LIN {X 0,Y 736.002,Z 322.542,A -85,B 0,C 180,E1 27536.573,E2 27536.573} C_VEL
LIN {X 0,Y 736.007,Z 322.537,A -85,B 0,C 180,E1 27534.23,E2 27534.23} C_VEL
LIN {X 0,Y 736.096,Z 322.542,A -85,B 0,C 180,E1 27531.444,E2 27531.444} C_VEL
LIN {X 0,Y 736.087,Z 322.537,A -85,B 0,C 180,E1 27529.14,E2 27529.14} C_VEL
LIN {X 0,Y 735.045,Z 322.662,A -85,B 0,C 180,E1 27528.541,E2 27528.541} C_VEL
LIN {X 0,Y 728.618,Z 323.468,A -85,B 0,C 180,E1 27526.861,E2 27526.861} C_VEL
LIN {X 0,Y 728.077,Z 323.53,A -85,B 0,C 180,E1 27526.425,E2 27526.425} C_VEL
LIN {X 0,Y 728.078,Z 323.523,A -85,B 0,C 180,E1 27524.01,E2 27524.01} C_VEL
LIN {X 0,Y 728.156,Z 323.53,A -85,B 0,C 180,E1 27521.257,E2 27521.257} C_VEL
LIN {X 0,Y 728.092,Z 323.528,A -85,B 0,C 180,E1 27518.389,E2 27518.389} C_VEL
LIN {X 0,Y 728.082,Z 323.529,A -85,B 0,C 180,E1 27515.928,E2 27515.928} C_VEL
LIN {X 0,Y 728.15,Z 323.533,A -85,B 0,C 180,E1 27513.196,E2 27513.196} C_VEL
LIN {X 0,Y 728.1,Z 323.527,A -85,B 0,C 180,E1 27510.215,E2 27510.215} C_VEL
LIN {X 0,Y 728.091,Z 323.531,A -85,B 0,C 180,E1 27507.709,E2 27507.709} C_VEL
LIN {X 0,Y 728.156,Z 323.534,A -85,B 0,C 180,E1 27504.925,E2 27504.925} C_VEL
LIN {X 0,Y 728.109,Z 323.531,A -85,B 0,C 180,E1 27502.021,E2 27502.021} C_VEL
LIN {X 0,Y 728.178,Z 323.766,A -85,B 0,C 180,E1 27500.292,E2 27500.292} C_VEL
LIN {X 0,Y 729.309,Z 326.852,A -85,B 0,C 180,E1 27499.984,E2 27499.984} C_VEL
LIN {X 0,Y 733.452,Z 336.015,A -85,B 0,C 180,E1 27499.025,E2 27499.025} C_VEL
LIN {X 0,Y 733.504,Z 341.36,A -85,B 0,C 180,E1 27498.676,E2 27498.676} C_VEL
LIN {X 0,Y 735.856,Z 350.593,A -85,B 0,C 180,E1 27498.388,E2 27498.388} C_VEL
LIN {X 0,Y 734.928,Z 566.12,A -85,B 0,C 180,E1 27495.714,E2 27495.714} C_VEL
LIN {X 0,Y 734.028,Z 793.03,A -85,B 0,C 180,E1 27492.997,E2 27492.997} C_VEL
LIN {X 0,Y 733.826,Z 825.795,A -85,B 0,C 180,E1 27492.567,E2 27492.567} C_VEL
LIN {X 0,Y 733.495,Z 853.318,A -85,B 0,C 180,E1 27492.041,E2 27492.041} C_VEL
LIN {X 0,Y 733.131,Z 879.099,A -85,B 0,C 180,E1 27491.393,E2 27491.393} C_VEL
LIN {X 0,Y 732.64,Z 907.823,A -85,B 0,C 180,E1 27490.487,E2 27490.487} C_VEL
LIN {X 0,Y 732.19,Z 930.681,A -85,B 0,C 180,E1 27489.622,E2 27489.622} C_VEL
LIN {X 0,Y 731.795,Z 951.079,A -85,B 0,C 180,E1 27488.739,E2 27488.739} C_VEL
LIN {X 0,Y 731.381,Z 971.985,A -85,B 0,C 180,E1 27487.718,E2 27487.718} C_VEL
LIN {X 0,Y 730.845,Z 997.329,A -85,B 0,C 180,E1 27486.309,E2 27486.309} C_VEL
LIN {X 0,Y 730.379,Z 1017.32,A -85,B 0,C 180,E1 27485.048,E2 27485.048} C_VEL
LIN {X 0,Y 730.011,Z 1035.431,A -85,B 0,C 180,E1 27483.785,E2 27483.785} C_VEL
LIN {X 0,Y 729.644,Z 1055.852,A -85,B 0,C 180,E1 27482.213,E2 27482.213} C_VEL
LIN {X 0,Y 729.213,Z 1074.861,A -85,B 0,C 180,E1 27480.558,E2 27480.558} C_VEL
LIN {X 0,Y 728.957,Z 1090.57,A -85,B 0,C 180,E1 27479.049,E2 27479.049} C_VEL
LIN {X 0,Y 728.689,Z 1108.03,A -85,B 0,C 180,E1 27477.189,E2 27477.189} C_VEL
LIN {X 0,Y 728.436,Z 1123.152,A -85,B 0,C 180,E1 27475.357,E2 27475.357} C_VEL
LIN {X 0,Y 728.291,Z 1134.68,A -85,B 0,C 180,E1 27473.805,E2 27473.805} C_VEL
LIN {X 0,Y 728.159,Z 1145.498,A -85,B 0,C 180,E1 27472.186,E2 27472.186} C_VEL
LIN {X 0,Y 728.088,Z 1156.487,A -85,B 0,C 180,E1 27470.331,E2 27470.331} C_VEL
LIN {X 0,Y 727.975,Z 1167.358,A -85,B 0,C 180,E1 27468.166,E2 27468.166} C_VEL
LIN {X 0,Y 727.957,Z 1175.727,A -85,B 0,C 180,E1 27466.19,E2 27466.19} C_VEL
LIN {X 0,Y 727.928,Z 1182.921,A -85,B 0,C 180,E1 27464.071,E2 27464.071} C_VEL
LIN {X 0,Y 727.913,Z 1188.371,A -85,B 0,C 180,E1 27461.971,E2 27461.971} C_VEL
LIN {X 0,Y 727.907,Z 1192.173,A -85,B 0,C 180,E1 27459.887,E2 27459.887} C_VEL
LIN {X 0,Y 727.904,Z 1194.402,A -85,B 0,C 180,E1 27457.736,E2 27457.736} C_VEL
LIN {X 0,Y 727.892,Z 1194.882,A -85,B 0,C 180,E1 27455.518,E2 27455.518} C_VEL
LIN {X 0,Y 727.906,Z 1193.93,A -85,B 0,C 180,E1 27453.544,E2 27453.544} C_VEL
LIN {X 0,Y 727.907,Z 1191.228,A -85,B 0,C 180,E1 27451.416,E2 27451.416} C_VEL
LIN {X 0,Y 727.917,Z 1187.057,A -85,B 0,C 180,E1 27449.37,E2 27449.37} C_VEL
LIN {X 0,Y 727.937,Z 1181.082,A -85,B 0,C 180,E1 27447.244,E2 27447.244} C_VEL
LIN {X 0,Y 727.952,Z 1173.342,A -85,B 0,C 180,E1 27445.114,E2 27445.114} C_VEL
LIN {X 0,Y 728.022,Z 1163.33,A -85,B 0,C 180,E1 27442.899,E2 27442.899} C_VEL
LIN {X 0,Y 728.076,Z 1154.04,A -85,B 0,C 180,E1 27441.152,E2 27441.152} C_VEL
LIN {X 0,Y 728.191,Z 1144.427,A -85,B 0,C 180,E1 27439.557,E2 27439.557} C_VEL
LIN {X 0,Y 728.307,Z 1133.054,A -85,B 0,C 180,E1 27437.874,E2 27437.874} C_VEL
LIN {X 0,Y 728.521,Z 1117.682,A -85,B 0,C 180,E1 27435.859,E2 27435.859} C_VEL
LIN {X 0,Y 728.753,Z 1102.122,A -85,B 0,C 180,E1 27434.073,E2 27434.073} C_VEL
LIN {X 0,Y 728.985,Z 1087.151,A -85,B 0,C 180,E1 27432.519,E2 27432.519} C_VEL
LIN {X 0,Y 729.387,Z 1068.169,A -85,B 0,C 180,E1 27430.745,E2 27430.745} C_VEL
LIN {X 0,Y 729.694,Z 1049.723,A -85,B 0,C 180,E1 27429.212,E2 27429.212} C_VEL
LIN {X 0,Y 730.068,Z 1032.568,A -85,B 0,C 180,E1 27427.917,E2 27427.917} C_VEL
LIN {X 0,Y 730.59,Z 1011.035,A -85,B 0,C 180,E1 27426.445,E2 27426.445} C_VEL
LIN {X 0,Y 731.026,Z 987.732,A -85,B 0,C 180,E1 27425.046,E2 27425.046} C_VEL
LIN {X 0,Y 731.424,Z 968.525,A -85,B 0,C 180,E1 27424.015,E2 27424.015} C_VEL
LIN {X 0,Y 731.828,Z 948.858,A -85,B 0,C 180,E1 27423.069,E2 27423.069} C_VEL
LIN {X 0,Y 732.349,Z 925.446,A -85,B 0,C 180,E1 27422.076,E2 27422.076} C_VEL
LIN {X 0,Y 732.817,Z 899.396,A -85,B 0,C 180,E1 27421.14,E2 27421.14} C_VEL
LIN {X 0,Y 733.19,Z 875.306,A -85,B 0,C 180,E1 27420.412,E2 27420.412} C_VEL
LIN {X 0,Y 733.552,Z 848.854,A -85,B 0,C 180,E1 27419.773,E2 27419.773} C_VEL
LIN {X 0,Y 733.842,Z 821.735,A -85,B 0,C 180,E1 27419.281,E2 27419.281} C_VEL
LIN {X 0,Y 734.101,Z 774.815,A -85,B 0,C 180,E1 27418.699,E2 27418.699} C_VEL
LIN {X 0,Y 734.997,Z 548.599,A -85,B 0,C 180,E1 27415.982,E2 27415.982} C_VEL
LIN {X 0,Y 735.843,Z 349.755,A -85,B 0,C 180,E1 27413.511,E2 27413.511} C_VEL
LIN {X 0,Y 733.426,Z 340.384,A -85,B 0,C 180,E1 27413.189,E2 27413.189} C_VEL
LIN {X 0,Y 733.459,Z 336.113,A -85,B 0,C 180,E1 27412.893,E2 27412.893} C_VEL
LIN {X 0,Y 729.199,Z 326.593,A -85,B 0,C 180,E1 27411.9,E2 27411.9} C_VEL
LIN {X 0,Y 728.144,Z 323.532,A -85,B 0,C 180,E1 27411.584,E2 27411.584} C_VEL
LIN {X 0,Y 728.135,Z 323.53,A -85,B 0,C 180,E1 27408.691,E2 27408.691} C_VEL
LIN {X 0,Y 728.16,Z 323.524,A -85,B 0,C 180,E1 27405.768,E2 27405.768} C_VEL
LIN {X 0,Y 728.142,Z 323.533,A -85,B 0,C 180,E1 27402.716,E2 27402.716} C_VEL
LIN {X 0,Y 728.143,Z 323.524,A -85,B 0,C 180,E1 27399.786,E2 27399.786} C_VEL
LIN {X 0,Y 728.147,Z 323.533,A -85,B 0,C 180,E1 27396.68,E2 27396.68} C_VEL
LIN {X 0,Y 728.122,Z 323.525,A -85,B 0,C 180,E1 27393.819,E2 27393.819} C_VEL
LIN {X 0,Y 728.156,Z 323.531,A -85,B 0,C 180,E1 27390.882,E2 27390.882} C_VEL
LIN {X 0,Y 728.109,Z 323.526,A -85,B 0,C 180,E1 27388.101,E2 27388.101} C_VEL
LIN {X 0,Y 728.139,Z 323.518,A -85,B 0,C 180,E1 27385.369,E2 27385.369} C_VEL
LIN {X 0,Y 728.122,Z 323.528,A -85,B 0,C 180,E1 27382.273,E2 27382.273} C_VEL
LIN {X 0,Y 728.103,Z 323.52,A -85,B 0,C 180,E1 27379.578,E2 27379.578} C_VEL
LIN {X 0,Y 728.159,Z 323.529,A -85,B 0,C 180,E1 27376.678,E2 27376.678} C_VEL
LIN {X 0,Y 728.096,Z 323.52,A -85,B 0,C 180,E1 27373.854,E2 27373.854} C_VEL
LIN {X 0,Y 728.105,Z 323.526,A -85,B 0,C 180,E1 27371.245,E2 27371.245} C_VEL
LIN {X 0,Y 728.138,Z 323.533,A -85,B 0,C 180,E1 27368.211,E2 27368.211} C_VEL
LIN {X 0,Y 728.082,Z 323.528,A -85,B 0,C 180,E1 27365.517,E2 27365.517} C_VEL
LIN {X 0,Y 728.103,Z 323.528,A -85,B 0,C 180,E1 27362.991,E2 27362.991} C_VEL
LIN {X 0,Y 728.113,Z 323.533,A -85,B 0,C 180,E1 27359.921,E2 27359.921} C_VEL
LIN {X 0,Y 728.074,Z 323.531,A -85,B 0,C 180,E1 27357.402,E2 27357.402} C_VEL
LIN {X 0,Y 728.08,Z 323.529,A -85,B 0,C 180,E1 27354.958,E2 27354.958} C_VEL
LIN {X 0,Y 728.149,Z 323.531,A -85,B 0,C 180,E1 27352.028,E2 27352.028} C_VEL
LIN {X 0,Y 728.068,Z 323.532,A -85,B 0,C 180,E1 27349.315,E2 27349.315} C_VEL
LIN {X 0,Y 728.06,Z 323.525,A -85,B 0,C 180,E1 27346.983,E2 27346.983} C_VEL
LIN {X 0,Y 728.083,Z 323.529,A -85,B 0,C 180,E1 27344.548,E2 27344.548} C_VEL
LIN {X 0,Y 728.077,Z 323.527,A -85,B 0,C 180,E1 27341.421,E2 27341.421} C_VEL
LIN {X 0,Y 728.05,Z 323.531,A -85,B 0,C 180,E1 27338.995,E2 27338.995} C_VEL
LIN {X 0,Y 728.048,Z 323.534,A -85,B 0,C 180,E1 27336.749,E2 27336.749} C_VEL
LIN {X 0,Y 728.078,Z 323.524,A -85,B 0,C 180,E1 27334.276,E2 27334.276} C_VEL
LIN {X 0,Y 728.074,Z 323.533,A -85,B 0,C 180,E1 27331.181,E2 27331.181} C_VEL
LIN {X 0,Y 728.057,Z 323.531,A -85,B 0,C 180,E1 27328.818,E2 27328.818} C_VEL
LIN {X 0,Y 728.061,Z 323.534,A -85,B 0,C 180,E1 27326.472,E2 27326.472} C_VEL
LIN {X 0,Y 728.129,Z 323.535,A -85,B 0,C 180,E1 27323.808,E2 27323.808} C_VEL
LIN {X 0,Y 728.083,Z 323.535,A -85,B 0,C 180,E1 27320.888,E2 27320.888} C_VEL
LIN {X 0,Y 728.069,Z 323.533,A -85,B 0,C 180,E1 27318.446,E2 27318.446} C_VEL
LIN {X 0,Y 728.093,Z 323.537,A -85,B 0,C 180,E1 27315.981,E2 27315.981} C_VEL
LIN {X 0,Y 728.144,Z 323.69,A -85,B 0,C 180,E1 27315.022,E2 27315.022} C_VEL
LIN {X 0,Y 729.555,Z 327.257,A -85,B 0,C 180,E1 27314.658,E2 27314.658} C_VEL
LIN {X 0,Y 733.674,Z 336.351,A -85,B 0,C 180,E1 27313.706,E2 27313.706} C_VEL
LIN {X 0,Y 733.608,Z 351.232,A -85,B 0,C 180,E1 27312.715,E2 27312.715} C_VEL
LIN {X 0,Y 735.832,Z 360.077,A -85,B 0,C 180,E1 27312.441,E2 27312.441} C_VEL
LIN {X 0,Y 734.945,Z 570.243,A -85,B 0,C 180,E1 27309.832,E2 27309.832} C_VEL
LIN {X 0,Y 734.062,Z 795.119,A -85,B 0,C 180,E1 27307.135,E2 27307.135} C_VEL
LIN {X 0,Y 733.838,Z 833.798,A -85,B 0,C 180,E1 27306.643,E2 27306.643} C_VEL
LIN {X 0,Y 733.521,Z 860.678,A -85,B 0,C 180,E1 27306.143,E2 27306.143} C_VEL
LIN {X 0,Y 733.18,Z 886.466,A -85,B 0,C 180,E1 27305.512,E2 27305.512} C_VEL
LIN {X 0,Y 732.754,Z 914.371,A -85,B 0,C 180,E1 27304.654,E2 27304.654} C_VEL
LIN {X 0,Y 732.218,Z 939.469,A -85,B 0,C 180,E1 27303.717,E2 27303.717} C_VEL
LIN {X 0,Y 731.801,Z 960.579,A -85,B 0,C 180,E1 27302.808,E2 27302.808} C_VEL
LIN {X 0,Y 731.386,Z 982.079,A -85,B 0,C 180,E1 27301.758,E2 27301.758} C_VEL
LIN {X 0,Y 730.853,Z 1007.148,A -85,B 0,C 180,E1 27300.366,E2 27300.366} C_VEL
LIN {X 0,Y 730.377,Z 1027.561,A -85,B 0,C 180,E1 27299.078,E2 27299.078} C_VEL
LIN {X 0,Y 729.986,Z 1046.46,A -85,B 0,C 180,E1 27297.756,E2 27297.756} C_VEL
LIN {X 0,Y 729.574,Z 1068.227,A -85,B 0,C 180,E1 27296.056,E2 27296.056} C_VEL
LIN {X 0,Y 729.193,Z 1085.444,A -85,B 0,C 180,E1 27294.55,E2 27294.55} C_VEL
LIN {X 0,Y 728.946,Z 1101.387,A -85,B 0,C 180,E1 27293.012,E2 27293.012} C_VEL
LIN {X 0,Y 728.632,Z 1120.118,A -85,B 0,C 180,E1 27290.988,E2 27290.988} C_VEL
LIN {X 0,Y 728.422,Z 1133.8,A -85,B 0,C 180,E1 27289.318,E2 27289.318} C_VEL
LIN {X 0,Y 728.291,Z 1145.415,A -85,B 0,C 180,E1 27287.746,E2 27287.746} C_VEL
LIN {X 0,Y 728.151,Z 1156.938,A -85,B 0,C 180,E1 27286.005,E2 27286.005} C_VEL
LIN {X 0,Y 728.048,Z 1169.419,A -85,B 0,C 180,E1 27283.826,E2 27283.826} C_VEL
LIN {X 0,Y 727.974,Z 1178.071,A -85,B 0,C 180,E1 27282.051,E2 27282.051} C_VEL
LIN {X 0,Y 727.953,Z 1185.836,A -85,B 0,C 180,E1 27280.206,E2 27280.206} C_VEL
LIN {X 0,Y 727.927,Z 1193.11,A -85,B 0,C 180,E1 27278.054,E2 27278.054} C_VEL
LIN {X 0,Y 727.914,Z 1198.421,A -85,B 0,C 180,E1 27275.993,E2 27275.993} C_VEL
LIN {X 0,Y 727.907,Z 1202.277,A -85,B 0,C 180,E1 27273.86,E2 27273.86} C_VEL
LIN {X 0,Y 727.908,Z 1204.493,A -85,B 0,C 180,E1 27271.653,E2 27271.653} C_VEL
LIN {X 0,Y 727.89,Z 1204.872,A -85,B 0,C 180,E1 27269.528,E2 27269.528} C_VEL
LIN {X 0,Y 727.906,Z 1203.905,A -85,B 0,C 180,E1 27267.56,E2 27267.56} C_VEL
LIN {X 0,Y 727.907,Z 1201.179,A -85,B 0,C 180,E1 27265.431,E2 27265.431} C_VEL
LIN {X 0,Y 727.916,Z 1196.957,A -85,B 0,C 180,E1 27263.375,E2 27263.375} C_VEL
LIN {X 0,Y 727.936,Z 1191.149,A -85,B 0,C 180,E1 27261.31,E2 27261.31} C_VEL
LIN {X 0,Y 727.945,Z 1183.639,A -85,B 0,C 180,E1 27259.234,E2 27259.234} C_VEL
LIN {X 0,Y 728.028,Z 1173.527,A -85,B 0,C 180,E1 27256.983,E2 27256.983} C_VEL
LIN {X 0,Y 728.084,Z 1164.528,A -85,B 0,C 180,E1 27255.282,E2 27255.282} C_VEL
LIN {X 0,Y 728.169,Z 1154.742,A -85,B 0,C 180,E1 27253.651,E2 27253.651} C_VEL
LIN {X 0,Y 728.298,Z 1144.115,A -85,B 0,C 180,E1 27252.07,E2 27252.07} C_VEL
LIN {X 0,Y 728.489,Z 1130.976,A -85,B 0,C 180,E1 27250.318,E2 27250.318} C_VEL
LIN {X 0,Y 728.741,Z 1113.473,A -85,B 0,C 180,E1 27248.264,E2 27248.264} C_VEL
LIN {X 0,Y 728.956,Z 1098.833,A -85,B 0,C 180,E1 27246.732,E2 27246.732} C_VEL
LIN {X 0,Y 729.278,Z 1082.528,A -85,B 0,C 180,E1 27245.183,E2 27245.183} C_VEL
LIN {X 0,Y 729.687,Z 1061.272,A -85,B 0,C 180,E1 27243.38,E2 27243.38} C_VEL
LIN {X 0,Y 730.037,Z 1043.447,A -85,B 0,C 180,E1 27242.025,E2 27242.025} C_VEL
LIN {X 0,Y 730.495,Z 1023.595,A -85,B 0,C 180,E1 27240.659,E2 27240.659} C_VEL
LIN {X 0,Y 731.011,Z 999.737,A -85,B 0,C 180,E1 27239.204,E2 27239.204} C_VEL
LIN {X 0,Y 731.426,Z 978.531,A -85,B 0,C 180,E1 27238.06,E2 27238.06} C_VEL
LIN {X 0,Y 731.863,Z 957.714,A -85,B 0,C 180,E1 27237.061,E2 27237.061} C_VEL
LIN {X 0,Y 732.437,Z 932.727,A -85,B 0,C 180,E1 27236.012,E2 27236.012} C_VEL
LIN {X 0,Y 732.844,Z 907.023,A -85,B 0,C 180,E1 27235.109,E2 27235.109} C_VEL
LIN {X 0,Y 733.217,Z 883.762,A -85,B 0,C 180,E1 27234.416,E2 27234.416} C_VEL
LIN {X 0,Y 733.575,Z 857.292,A -85,B 0,C 180,E1 27233.785,E2 27233.785} C_VEL
LIN {X 0,Y 733.854,Z 830.083,A -85,B 0,C 180,E1 27233.3,E2 27233.3} C_VEL
LIN {X 0,Y 734.247,Z 744.981,A -85,B 0,C 180,E1 27232.271,E2 27232.271} C_VEL
LIN {X 0,Y 735.141,Z 523.003,A -85,B 0,C 180,E1 27229.59,E2 27229.59} C_VEL
LIN {X 0,Y 735.76,Z 359.115,A -85,B 0,C 180,E1 27227.541,E2 27227.541} C_VEL
LIN {X 0,Y 733.481,Z 350.368,A -85,B 0,C 180,E1 27227.245,E2 27227.245} C_VEL
LIN {X 0,Y 733.541,Z 335.961,A -85,B 0,C 180,E1 27226.257,E2 27226.257} C_VEL
LIN {X 0,Y 728.192,Z 324.004,A -85,B 0,C 180,E1 27225.004,E2 27225.004} C_VEL
LIN {X 0,Y 728.129,Z 323.534,A -85,B 0,C 180,E1 27224.943,E2 27224.943} C_VEL
LIN {X 0,Y 728.093,Z 323.536,A -85,B 0,C 180,E1 27221.975,E2 27221.975} C_VEL
LIN {X 0,Y 728.069,Z 323.534,A -85,B 0,C 180,E1 27219.484,E2 27219.484} C_VEL
LIN {X 0,Y 728.082,Z 323.532,A -85,B 0,C 180,E1 27217.072,E2 27217.072} C_VEL
LIN {X 0,Y 728.128,Z 323.533,A -85,B 0,C 180,E1 27214.102,E2 27214.102} C_VEL
LIN {X 0,Y 728.065,Z 323.53,A -85,B 0,C 180,E1 27211.458,E2 27211.458} C_VEL
LIN {X 0,Y 728.058,Z 323.532,A -85,B 0,C 180,E1 27209.18,E2 27209.18} C_VEL
LIN {X 0,Y 728.069,Z 323.53,A -85,B 0,C 180,E1 27206.861,E2 27206.861} C_VEL
LIN {X 0,Y 728.138,Z 323.534,A -85,B 0,C 180,E1 27203.984,E2 27203.984} C_VEL
LIN {X 0,Y 728.059,Z 323.529,A -85,B 0,C 180,E1 27201.343,E2 27201.343} C_VEL
LIN {X 0,Y 728.05,Z 323.534,A -85,B 0,C 180,E1 27198.995,E2 27198.995} C_VEL
LIN {X 0,Y 728.06,Z 323.528,A -85,B 0,C 180,E1 27196.598,E2 27196.598} C_VEL
LIN {X 0,Y 728.117,Z 323.533,A -85,B 0,C 180,E1 27193.662,E2 27193.662} C_VEL
LIN {X 0,Y 728.052,Z 323.527,A -85,B 0,C 180,E1 27191.005,E2 27191.005} C_VEL
LIN {X 0,Y 728.05,Z 323.534,A -85,B 0,C 180,E1 27188.689,E2 27188.689} C_VEL
LIN {X 0,Y 728.073,Z 323.53,A -85,B 0,C 180,E1 27186.308,E2 27186.308} C_VEL
LIN {X 0,Y 728.106,Z 323.532,A -85,B 0,C 180,E1 27183.293,E2 27183.293} C_VEL
LIN {X 0,Y 728.06,Z 323.525,A -85,B 0,C 180,E1 27180.708,E2 27180.708} C_VEL
LIN {X 0,Y 728.062,Z 323.531,A -85,B 0,C 180,E1 27178.426,E2 27178.426} C_VEL
LIN {X 0,Y 728.1,Z 323.533,A -85,B 0,C 180,E1 27175.905,E2 27175.905} C_VEL
LIN {X 0,Y 728.096,Z 323.53,A -85,B 0,C 180,E1 27172.9,E2 27172.9} C_VEL
LIN {X 0,Y 728.07,Z 323.528,A -85,B 0,C 180,E1 27170.415,E2 27170.415} C_VEL
LIN {X 0,Y 728.079,Z 323.529,A -85,B 0,C 180,E1 27168.032,E2 27168.032} C_VEL
LIN {X 0,Y 728.077,Z 323.53,A -85,B 0,C 180,E1 27166.425,E2 27166.425} C_VEL
LIN {X 0,Y 727.066,Z 323.662,A -85,B 0,C 180,E1 27165.819,E2 27165.819} C_VEL
LIN {X 0,Y 720.656,Z 324.446,A -85,B 0,C 180,E1 27164.12,E2 27164.12} C_VEL
LIN {X 0,Y 720.166,Z 324.511,A -85,B 0,C 180,E1 27163.679,E2 27163.679} C_VEL
LIN {X 0,Y 720.169,Z 324.512,A -85,B 0,C 180,E1 27160.62,E2 27160.62} C_VEL
LIN {X 0,Y 720.141,Z 324.519,A -85,B 0,C 180,E1 27158.044,E2 27158.044} C_VEL
LIN {X 0,Y 720.184,Z 324.516,A -85,B 0,C 180,E1 27155.385,E2 27155.385} C_VEL
LIN {X 0,Y 720.169,Z 324.516,A -85,B 0,C 180,E1 27152.348,E2 27152.348} C_VEL
LIN {X 0,Y 720.149,Z 324.518,A -85,B 0,C 180,E1 27149.826,E2 27149.826} C_VEL
LIN {X 0,Y 720.203,Z 324.523,A -85,B 0,C 180,E1 27147.122,E2 27147.122} C_VEL
LIN {X 0,Y 720.174,Z 324.52,A -85,B 0,C 180,E1 27144.133,E2 27144.133} C_VEL
LIN {X 0,Y 720.16,Z 324.524,A -85,B 0,C 180,E1 27141.536,E2 27141.536} C_VEL
LIN {X 0,Y 720.239,Z 324.675,A -85,B 0,C 180,E1 27140.845,E2 27140.845} C_VEL
LIN {X 0,Y 721.528,Z 328.003,A -85,B 0,C 180,E1 27140.5,E2 27140.5} C_VEL
LIN {X 0,Y 726.876,Z 340.375,A -85,B 0,C 180,E1 27139.201,E2 27139.201} C_VEL
LIN {X 0,Y 729.929,Z 352.779,A -85,B 0,C 180,E1 27138.786,E2 27138.786} C_VEL
LIN {X 0,Y 728.752,Z 569.074,A -85,B 0,C 180,E1 27136.082,E2 27136.082} C_VEL
LIN {X 0,Y 727.619,Z 796.028,A -85,B 0,C 180,E1 27133.342,E2 27133.342} C_VEL
LIN {X 0,Y 727.36,Z 826.961,A -85,B 0,C 180,E1 27132.926,E2 27132.926} C_VEL
LIN {X 0,Y 726.951,Z 854.16,A -85,B 0,C 180,E1 27132.397,E2 27132.397} C_VEL
LIN {X 0,Y 726.506,Z 879.854,A -85,B 0,C 180,E1 27131.744,E2 27131.744} C_VEL
LIN {X 0,Y 725.901,Z 908.235,A -85,B 0,C 180,E1 27130.838,E2 27130.838} C_VEL
LIN {X 0,Y 725.375,Z 929.832,A -85,B 0,C 180,E1 27130.018,E2 27130.018} C_VEL
LIN {X 0,Y 724.855,Z 950.312,A -85,B 0,C 180,E1 27129.13,E2 27129.13} C_VEL
LIN {X 0,Y 724.32,Z 971.291,A -85,B 0,C 180,E1 27128.101,E2 27128.101} C_VEL
LIN {X 0,Y 723.688,Z 996.404,A -85,B 0,C 180,E1 27126.7,E2 27126.7} C_VEL
LIN {X 0,Y 723.094,Z 1016.788,A -85,B 0,C 180,E1 27125.407,E2 27125.407} C_VEL
LIN {X 0,Y 722.602,Z 1034.953,A -85,B 0,C 180,E1 27124.131,E2 27124.131} C_VEL
LIN {X 0,Y 722.133,Z 1054.845,A -85,B 0,C 180,E1 27122.589,E2 27122.589} C_VEL
LIN {X 0,Y 721.611,Z 1074.295,A -85,B 0,C 180,E1 27120.888,E2 27120.888} C_VEL
LIN {X 0,Y 721.251,Z 1089.79,A -85,B 0,C 180,E1 27119.39,E2 27119.39} C_VEL
LIN {X 0,Y 720.929,Z 1106.602,A -85,B 0,C 180,E1 27117.592,E2 27117.592} C_VEL
LIN {X 0,Y 720.597,Z 1122.573,A -85,B 0,C 180,E1 27115.653,E2 27115.653} C_VEL
LIN {X 0,Y 720.398,Z 1134.766,A -85,B 0,C 180,E1 27113.995,E2 27113.995} C_VEL
LIN {X 0,Y 720.231,Z 1145.577,A -85,B 0,C 180,E1 27112.357,E2 27112.357} C_VEL
LIN {X 0,Y 720.136,Z 1156.558,A -85,B 0,C 180,E1 27110.48,E2 27110.48} C_VEL
LIN {X 0,Y 720.007,Z 1167.416,A -85,B 0,C 180,E1 27108.291,E2 27108.291} C_VEL
LIN {X 0,Y 719.97,Z 1175.772,A -85,B 0,C 180,E1 27106.292,E2 27106.292} C_VEL
LIN {X 0,Y 719.932,Z 1182.961,A -85,B 0,C 180,E1 27104.148,E2 27104.148} C_VEL
LIN {X 0,Y 719.914,Z 1188.4,A -85,B 0,C 180,E1 27102.024,E2 27102.024} C_VEL
LIN {X 0,Y 719.907,Z 1192.19,A -85,B 0,C 180,E1 27099.917,E2 27099.917} C_VEL
LIN {X 0,Y 719.904,Z 1194.411,A -85,B 0,C 180,E1 27097.742,E2 27097.742} C_VEL
LIN {X 0,Y 719.891,Z 1194.9,A -85,B 0,C 180,E1 27095.579,E2 27095.579} C_VEL
LIN {X 0,Y 719.908,Z 1193.984,A -85,B 0,C 180,E1 27093.583,E2 27093.583} C_VEL
LIN {X 0,Y 719.908,Z 1191.332,A -85,B 0,C 180,E1 27091.432,E2 27091.432} C_VEL
LIN {X 0,Y 719.919,Z 1187.219,A -85,B 0,C 180,E1 27089.363,E2 27089.363} C_VEL
LIN {X 0,Y 719.942,Z 1181.29,A -85,B 0,C 180,E1 27087.214,E2 27087.214} C_VEL
LIN {X 0,Y 719.963,Z 1173.922,A -85,B 0,C 180,E1 27085.14,E2 27085.14} C_VEL
LIN {X 0,Y 720.055,Z 1163.673,A -85,B 0,C 180,E1 27082.82,E2 27082.82} C_VEL
LIN {X 0,Y 720.125,Z 1154.43,A -85,B 0,C 180,E1 27081.053,E2 27081.053} C_VEL
LIN {X 0,Y 720.263,Z 1144.484,A -85,B 0,C 180,E1 27079.38,E2 27079.38} C_VEL
LIN {X 0,Y 720.442,Z 1132.976,A -85,B 0,C 180,E1 27077.659,E2 27077.659} C_VEL
LIN {X 0,Y 720.697,Z 1117.588,A -85,B 0,C 180,E1 27075.62,E2 27075.62} C_VEL
LIN {X 0,Y 720.978,Z 1102.027,A -85,B 0,C 180,E1 27073.814,E2 27073.814} C_VEL
LIN {X 0,Y 721.316,Z 1086.976,A -85,B 0,C 180,E1 27072.237,E2 27072.237} C_VEL
LIN {X 0,Y 721.786,Z 1067.375,A -85,B 0,C 180,E1 27070.392,E2 27070.392} C_VEL
LIN {X 0,Y 722.224,Z 1049.054,A -85,B 0,C 180,E1 27068.86,E2 27068.86} C_VEL
LIN {X 0,Y 722.726,Z 1031.261,A -85,B 0,C 180,E1 27067.509,E2 27067.509} C_VEL
LIN {X 0,Y 723.357,Z 1008.839,A -85,B 0,C 180,E1 27065.978,E2 27065.978} C_VEL
LIN {X 0,Y 723.867,Z 987.456,A -85,B 0,C 180,E1 27064.69,E2 27064.69} C_VEL
LIN {X 0,Y 724.414,Z 967.445,A -85,B 0,C 180,E1 27063.612,E2 27063.612} C_VEL
LIN {X 0,Y 725.019,Z 945.758,A -85,B 0,C 180,E1 27062.573,E2 27062.573} C_VEL
LIN {X 0,Y 725.679,Z 919.441,A -85,B 0,C 180,E1 27061.482,E2 27061.482} C_VEL
LIN {X 0,Y 726.149,Z 896.91,A -85,B 0,C 180,E1 27060.691,E2 27060.691} C_VEL
LIN {X 0,Y 726.611,Z 873.986,A -85,B 0,C 180,E1 27060.003,E2 27060.003} C_VEL
LIN {X 0,Y 727.088,Z 847.004,A -85,B 0,C 180,E1 27059.358,E2 27059.358} C_VEL
LIN {X 0,Y 727.413,Z 820.25,A -85,B 0,C 180,E1 27058.879,E2 27058.879} C_VEL
LIN {X 0,Y 727.864,Z 744.159,A -85,B 0,C 180,E1 27057.949,E2 27057.949} C_VEL
LIN {X 0,Y 728.945,Z 526.82,A -85,B 0,C 180,E1 27055.305,E2 27055.305} C_VEL
LIN {X 0,Y 729.854,Z 351.702,A -85,B 0,C 180,E1 27053.105,E2 27053.105} C_VEL
LIN {X 0,Y 726.921,Z 340.55,A -85,B 0,C 180,E1 27052.725,E2 27052.725} C_VEL
LIN {X 0,Y 721.508,Z 328.001,A -85,B 0,C 180,E1 27051.409,E2 27051.409} C_VEL
LIN {X 0,Y 720.219,Z 324.521,A -85,B 0,C 180,E1 27051.029,E2 27051.029} C_VEL
LIN {X 0,Y 720.207,Z 324.511,A -85,B 0,C 180,E1 27047.997,E2 27047.997} C_VEL
LIN {X 0,Y 720.218,Z 324.522,A -85,B 0,C 180,E1 27044.925,E2 27044.925} C_VEL
LIN {X 0,Y 720.191,Z 324.514,A -85,B 0,C 180,E1 27042.005,E2 27042.005} C_VEL
LIN {X 0,Y 720.213,Z 324.52,A -85,B 0,C 180,E1 27039.073,E2 27039.073} C_VEL
LIN {X 0,Y 720.179,Z 324.517,A -85,B 0,C 180,E1 27036.23,E2 27036.23} C_VEL
LIN {X 0,Y 720.22,Z 324.512,A -85,B 0,C 180,E1 27033.352,E2 27033.352} C_VEL
LIN {X 0,Y 720.184,Z 324.52,A -85,B 0,C 180,E1 27030.356,E2 27030.356} C_VEL
LIN {X 0,Y 720.19,Z 324.51,A -85,B 0,C 180,E1 27027.538,E2 27027.538} C_VEL
LIN {X 0,Y 720.199,Z 324.522,A -85,B 0,C 180,E1 27024.439,E2 27024.439} C_VEL
LIN {X 0,Y 720.164,Z 324.512,A -85,B 0,C 180,E1 27021.674,E2 27021.674} C_VEL
LIN {X 0,Y 720.219,Z 324.509,A -85,B 0,C 180,E1 27018.789,E2 27018.789} C_VEL
LIN {X 0,Y 720.163,Z 324.516,A -85,B 0,C 180,E1 27015.957,E2 27015.957} C_VEL
LIN {X 0,Y 720.164,Z 324.504,A -85,B 0,C 180,E1 27013.325,E2 27013.325} C_VEL
LIN {X 0,Y 720.208,Z 324.522,A -85,B 0,C 180,E1 27010.317,E2 27010.317} C_VEL
LIN {X 0,Y 720.147,Z 324.519,A -85,B 0,C 180,E1 27007.58,E2 27007.58} C_VEL
LIN {X 0,Y 720.166,Z 324.514,A -85,B 0,C 180,E1 27005.018,E2 27005.018} C_VEL
LIN {X 0,Y 720.169,Z 324.519,A -85,B 0,C 180,E1 27001.91,E2 27001.91} C_VEL
LIN {X 0,Y 720.137,Z 324.52,A -85,B 0,C 180,E1 26999.364,E2 26999.364} C_VEL
LIN {X 0,Y 720.152,Z 324.518,A -85,B 0,C 180,E1 26996.896,E2 26996.896} C_VEL
LIN {X 0,Y 720.178,Z 324.523,A -85,B 0,C 180,E1 26993.863,E2 26993.863} C_VEL
LIN {X 0,Y 720.127,Z 324.519,A -85,B 0,C 180,E1 26991.295,E2 26991.295} C_VEL
LIN {X 0,Y 720.127,Z 324.521,A -85,B 0,C 180,E1 26988.953,E2 26988.953} C_VEL
LIN {X 0,Y 720.205,Z 324.508,A -85,B 0,C 180,E1 26986.185,E2 26986.185} C_VEL
LIN {X 0,Y 720.126,Z 324.523,A -85,B 0,C 180,E1 26983.296,E2 26983.296} C_VEL
LIN {X 0,Y 720.113,Z 324.514,A -85,B 0,C 180,E1 26980.955,E2 26980.955} C_VEL
LIN {X 0,Y 720.12,Z 324.52,A -85,B 0,C 180,E1 26978.581,E2 26978.581} C_VEL
LIN {X 0,Y 720.2,Z 324.511,A -85,B 0,C 180,E1 26975.735,E2 26975.735} C_VEL
LIN {X 0,Y 720.117,Z 324.523,A -85,B 0,C 180,E1 26972.996,E2 26972.996} C_VEL
LIN {X 0,Y 720.114,Z 324.522,A -85,B 0,C 180,E1 26970.65,E2 26970.65} C_VEL
LIN {X 0,Y 720.138,Z 324.521,A -85,B 0,C 180,E1 26968.249,E2 26968.249} C_VEL
LIN {X 0,Y 720.163,Z 324.522,A -85,B 0,C 180,E1 26965.205,E2 26965.205} C_VEL
LIN {X 0,Y 720.127,Z 324.523,A -85,B 0,C 180,E1 26962.643,E2 26962.643} C_VEL
LIN {X 0,Y 720.134,Z 324.526,A -85,B 0,C 180,E1 26960.283,E2 26960.283} C_VEL
LIN {X 0,Y 720.218,Z 324.522,A -85,B 0,C 180,E1 26957.459,E2 26957.459} C_VEL
LIN {X 0,Y 720.208,Z 324.545,A -85,B 0,C 180,E1 26955.595,E2 26955.595} C_VEL
LIN {X 0,Y 721.468,Z 327.925,A -85,B 0,C 180,E1 26955.247,E2 26955.247} C_VEL
LIN {X 0,Y 727.142,Z 340.615,A -85,B 0,C 180,E1 26953.9,E2 26953.9} C_VEL
LIN {X 0,Y 727.071,Z 351.187,A -85,B 0,C 180,E1 26953.193,E2 26953.193} C_VEL
LIN {X 0,Y 729.903,Z 362.253,A -85,B 0,C 180,E1 26952.839,E2 26952.839} C_VEL
LIN {X 0,Y 728.781,Z 572.279,A -85,B 0,C 180,E1 26950.211,E2 26950.211} C_VEL
LIN {X 0,Y 727.668,Z 796.593,A -85,B 0,C 180,E1 26947.499,E2 26947.499} C_VEL
LIN {X 0,Y 727.391,Z 834.551,A -85,B 0,C 180,E1 26947.01,E2 26947.01} C_VEL
LIN {X 0,Y 726.988,Z 861.9,A -85,B 0,C 180,E1 26946.493,E2 26946.493} C_VEL
LIN {X 0,Y 726.557,Z 887.52,A -85,B 0,C 180,E1 26945.855,E2 26945.855} C_VEL
LIN {X 0,Y 725.975,Z 916.182,A -85,B 0,C 180,E1 26944.957,E2 26944.957} C_VEL
LIN {X 0,Y 725.377,Z 939.908,A -85,B 0,C 180,E1 26944.06,E2 26944.06} C_VEL
LIN {X 0,Y 724.836,Z 961.082,A -85,B 0,C 180,E1 26943.139,E2 26943.139} C_VEL
LIN {X 0,Y 724.297,Z 983.242,A -85,B 0,C 180,E1 26942.045,E2 26942.045} C_VEL
LIN {X 0,Y 723.607,Z 1008.61,A -85,B 0,C 180,E1 26940.61,E2 26940.61} C_VEL
LIN {X 0,Y 723.048,Z 1028.225,A -85,B 0,C 180,E1 26939.356,E2 26939.356} C_VEL
LIN {X 0,Y 722.541,Z 1047.293,A -85,B 0,C 180,E1 26938.005,E2 26938.005} C_VEL
LIN {X 0,Y 721.988,Z 1069.75,A -85,B 0,C 180,E1 26936.218,E2 26936.218} C_VEL
LIN {X 0,Y 721.544,Z 1086.376,A -85,B 0,C 180,E1 26934.74,E2 26934.74} C_VEL
LIN {X 0,Y 721.207,Z 1103.089,A -85,B 0,C 180,E1 26933.101,E2 26933.101} C_VEL
LIN {X 0,Y 720.819,Z 1120.831,A -85,B 0,C 180,E1 26931.141,E2 26931.141} C_VEL
LIN {X 0,Y 720.582,Z 1133.802,A -85,B 0,C 180,E1 26929.537,E2 26929.537} C_VEL
LIN {X 0,Y 720.389,Z 1145.999,A -85,B 0,C 180,E1 26927.863,E2 26927.863} C_VEL
LIN {X 0,Y 720.213,Z 1158.899,A -85,B 0,C 180,E1 26925.873,E2 26925.873} C_VEL
LIN {X 0,Y 720.079,Z 1170.241,A -85,B 0,C 180,E1 26923.818,E2 26923.818} C_VEL
LIN {X 0,Y 719.995,Z 1178.43,A -85,B 0,C 180,E1 26922.105,E2 26922.105} C_VEL
LIN {X 0,Y 719.966,Z 1186.133,A -85,B 0,C 180,E1 26920.24,E2 26920.24} C_VEL
LIN {X 0,Y 719.933,Z 1193.545,A -85,B 0,C 180,E1 26918.001,E2 26918.001} C_VEL
LIN {X 0,Y 719.917,Z 1198.936,A -85,B 0,C 180,E1 26915.819,E2 26915.819} C_VEL
LIN {X 0,Y 719.909,Z 1202.483,A -85,B 0,C 180,E1 26913.743,E2 26913.743} C_VEL
LIN {X 0,Y 719.909,Z 1204.549,A -85,B 0,C 180,E1 26911.592,E2 26911.592} C_VEL
LIN {X 0,Y 719.89,Z 1204.872,A -85,B 0,C 180,E1 26909.523,E2 26909.523} C_VEL
LIN {X 0,Y 719.906,Z 1203.902,A -85,B 0,C 180,E1 26907.533,E2 26907.533} C_VEL
LIN {X 0,Y 719.907,Z 1201.179,A -85,B 0,C 180,E1 26905.38,E2 26905.38} C_VEL
LIN {X 0,Y 719.916,Z 1196.833,A -85,B 0,C 180,E1 26903.249,E2 26903.249} C_VEL
LIN {X 0,Y 719.937,Z 1190.892,A -85,B 0,C 180,E1 26901.132,E2 26901.132} C_VEL
LIN {X 0,Y 719.972,Z 1183.001,A -85,B 0,C 180,E1 26898.951,E2 26898.951} C_VEL
LIN {X 0,Y 720.061,Z 1173.153,A -85,B 0,C 180,E1 26896.762,E2 26896.762} C_VEL
LIN {X 0,Y 720.128,Z 1164.065,A -85,B 0,C 180,E1 26895.034,E2 26895.034} C_VEL
LIN {X 0,Y 720.263,Z 1154.221,A -85,B 0,C 180,E1 26893.383,E2 26893.383} C_VEL
LIN {X 0,Y 720.441,Z 1142.511,A -85,B 0,C 180,E1 26891.637,E2 26891.637} C_VEL
LIN {X 0,Y 720.722,Z 1126.521,A -85,B 0,C 180,E1 26889.537,E2 26889.537} C_VEL
LIN {X 0,Y 720.991,Z 1111.843,A -85,B 0,C 180,E1 26887.839,E2 26887.839} C_VEL
LIN {X 0,Y 721.307,Z 1097.127,A -85,B 0,C 180,E1 26886.297,E2 26886.297} C_VEL
LIN {X 0,Y 721.784,Z 1077.879,A -85,B 0,C 180,E1 26884.481,E2 26884.481} C_VEL
LIN {X 0,Y 722.23,Z 1059.057,A -85,B 0,C 180,E1 26882.905,E2 26882.905} C_VEL
LIN {X 0,Y 722.736,Z 1041.027,A -85,B 0,C 180,E1 26881.537,E2 26881.537} C_VEL
LIN {X 0,Y 723.364,Z 1018.078,A -85,B 0,C 180,E1 26879.975,E2 26879.975} C_VEL
LIN {X 0,Y 723.901,Z 996.236,A -85,B 0,C 180,E1 26878.666,E2 26878.666} C_VEL
LIN {X 0,Y 724.473,Z 975.864,A -85,B 0,C 180,E1 26877.576,E2 26877.576} C_VEL
LIN {X 0,Y 725.164,Z 951.706,A -85,B 0,C 180,E1 26876.434,E2 26876.434} C_VEL
LIN {X 0,Y 725.714,Z 926.405,A -85,B 0,C 180,E1 26875.414,E2 26875.414} C_VEL
LIN {X 0,Y 726.174,Z 904.852,A -85,B 0,C 180,E1 26874.669,E2 26874.669} C_VEL
LIN {X 0,Y 726.647,Z 881.751,A -85,B 0,C 180,E1 26873.988,E2 26873.988} C_VEL
LIN {X 0,Y 727.127,Z 854.673,A -85,B 0,C 180,E1 26873.354,E2 26873.354} C_VEL
LIN {X 0,Y 727.45,Z 827.356,A -85,B 0,C 180,E1 26872.882,E2 26872.882} C_VEL
LIN {X 0,Y 728.658,Z 595.174,A -85,B 0,C 180,E1 26870.069,E2 26870.069} C_VEL
LIN {X 0,Y 729.734,Z 390.517,A -85,B 0,C 180,E1 26867.519,E2 26867.519} C_VEL
LIN {X 0,Y 729.733,Z 360.849,A -85,B 0,C 180,E1 26867.13,E2 26867.13} C_VEL
LIN {X 0,Y 726.958,Z 350.368,A -85,B 0,C 180,E1 26866.768,E2 26866.768} C_VEL
LIN {X 0,Y 727.029,Z 340.062,A -85,B 0,C 180,E1 26866.053,E2 26866.053} C_VEL
LIN {X 0,Y 721.468,Z 327.926,A -85,B 0,C 180,E1 26864.753,E2 26864.753} C_VEL
LIN {X 0,Y 720.204,Z 324.523,A -85,B 0,C 180,E1 26864.378,E2 26864.378} C_VEL
LIN {X 0,Y 720.135,Z 324.525,A -85,B 0,C 180,E1 26861.67,E2 26861.67} C_VEL
LIN {X 0,Y 720.138,Z 324.523,A -85,B 0,C 180,E1 26859.218,E2 26859.218} C_VEL
LIN {X 0,Y 720.22,Z 324.52,A -85,B 0,C 180,E1 26856.357,E2 26856.357} C_VEL
LIN {X 0,Y 720.129,Z 324.522,A -85,B 0,C 180,E1 26853.547,E2 26853.547} C_VEL
LIN {X 0,Y 720.123,Z 324.518,A -85,B 0,C 180,E1 26851.192,E2 26851.192} C_VEL
LIN {X 0,Y 720.151,Z 324.521,A -85,B 0,C 180,E1 26848.712,E2 26848.712} C_VEL
LIN {X 0,Y 720.146,Z 324.521,A -85,B 0,C 180,E1 26845.671,E2 26845.671} C_VEL
LIN {X 0,Y 720.116,Z 324.522,A -85,B 0,C 180,E1 26843.194,E2 26843.194} C_VEL
LIN {X 0,Y 720.114,Z 324.517,A -85,B 0,C 180,E1 26840.907,E2 26840.907} C_VEL
LIN {X 0,Y 720.171,Z 324.523,A -85,B 0,C 180,E1 26838.259,E2 26838.259} C_VEL
LIN {X 0,Y 720.123,Z 324.522,A -85,B 0,C 180,E1 26835.297,E2 26835.297} C_VEL
LIN {X 0,Y 720.108,Z 324.522,A -85,B 0,C 180,E1 26832.91,E2 26832.91} C_VEL
LIN {X 0,Y 720.117,Z 324.515,A -85,B 0,C 180,E1 26830.561,E2 26830.561} C_VEL
LIN {X 0,Y 720.217,Z 324.518,A -85,B 0,C 180,E1 26827.739,E2 26827.739} C_VEL
LIN {X 0,Y 720.124,Z 324.518,A -85,B 0,C 180,E1 26824.939,E2 26824.939} C_VEL
LIN {X 0,Y 720.12,Z 324.522,A -85,B 0,C 180,E1 26822.547,E2 26822.547} C_VEL
LIN {X 0,Y 720.148,Z 324.514,A -85,B 0,C 180,E1 26820.08,E2 26820.08} C_VEL
LIN {X 0,Y 720.151,Z 324.519,A -85,B 0,C 180,E1 26816.976,E2 26816.976} C_VEL
LIN {X 0,Y 720.125,Z 324.512,A -85,B 0,C 180,E1 26814.502,E2 26814.502} C_VEL
LIN {X 0,Y 720.138,Z 324.522,A -85,B 0,C 180,E1 26812.099,E2 26812.099} C_VEL
LIN {X 0,Y 720.215,Z 324.511,A -85,B 0,C 180,E1 26809.197,E2 26809.197} C_VEL
LIN {X 0,Y 720.139,Z 324.519,A -85,B 0,C 180,E1 26806.427,E2 26806.427} C_VEL
LIN {X 0,Y 720.138,Z 324.51,A -85,B 0,C 180,E1 26804.043,E2 26804.043} C_VEL
LIN {X 0,Y 720.166,Z 324.511,A -85,B 0,C 180,E1 26803.679,E2 26803.679} C_VEL
LIN {X 0,Y 719.242,Z 324.639,A -85,B 0,C 180,E1 26803.066,E2 26803.066} C_VEL
LIN {X 0,Y 712.745,Z 325.449,A -85,B 0,C 180,E1 26801.306,E2 26801.306} C_VEL
LIN {X 0,Y 712.267,Z 325.5,A -85,B 0,C 180,E1 26800.904,E2 26800.904} C_VEL
LIN {X 0,Y 712.205,Z 325.508,A -85,B 0,C 180,E1 26798.122,E2 26798.122} C_VEL
LIN {X 0,Y 712.228,Z 325.506,A -85,B 0,C 180,E1 26795.534,E2 26795.534} C_VEL
LIN {X 0,Y 712.236,Z 325.505,A -85,B 0,C 180,E1 26792.401,E2 26792.401} C_VEL
LIN {X 0,Y 712.21,Z 325.507,A -85,B 0,C 180,E1 26789.827,E2 26789.827} C_VEL
LIN {X 0,Y 712.269,Z 325.511,A -85,B 0,C 180,E1 26787.083,E2 26787.083} C_VEL
LIN {X 0,Y 712.23,Z 325.51,A -85,B 0,C 180,E1 26784.068,E2 26784.068} C_VEL
LIN {X 0,Y 712.245,Z 325.658,A -85,B 0,C 180,E1 26781.416,E2 26781.416} C_VEL
LIN {X 0,Y 713.753,Z 329.258,A -85,B 0,C 180,E1 26781.023,E2 26781.023} C_VEL
LIN {X 0,Y 719.216,Z 341.312,A -85,B 0,C 180,E1 26779.737,E2 26779.737} C_VEL
LIN {X 0,Y 721.673,Z 345.641,A -85,B 0,C 180,E1 26779.492,E2 26779.492} C_VEL
LIN {X 0,Y 724.035,Z 355.052,A -85,B 0,C 180,E1 26779.189,E2 26779.189} C_VEL
LIN {X 0,Y 722.608,Z 571.699,A -85,B 0,C 180,E1 26776.461,E2 26776.461} C_VEL
LIN {X 0,Y 721.238,Z 799.024,A -85,B 0,C 180,E1 26773.693,E2 26773.693} C_VEL
LIN {X 0,Y 720.903,Z 829.058,A -85,B 0,C 180,E1 26773.275,E2 26773.275} C_VEL
LIN {X 0,Y 720.432,Z 855.349,A -85,B 0,C 180,E1 26772.752,E2 26772.752} C_VEL
LIN {X 0,Y 719.89,Z 881.262,A -85,B 0,C 180,E1 26772.082,E2 26772.082} C_VEL
LIN {X 0,Y 719.163,Z 909.33,A -85,B 0,C 180,E1 26771.171,E2 26771.171} C_VEL
LIN {X 0,Y 718.569,Z 930.187,A -85,B 0,C 180,E1 26770.37,E2 26770.37} C_VEL
LIN {X 0,Y 717.945,Z 950.511,A -85,B 0,C 180,E1 26769.481,E2 26769.481} C_VEL
LIN {X 0,Y 717.277,Z 971.552,A -85,B 0,C 180,E1 26768.441,E2 26768.441} C_VEL
LIN {X 0,Y 716.526,Z 996.414,A -85,B 0,C 180,E1 26767.04,E2 26767.04} C_VEL
LIN {X 0,Y 715.808,Z 1016.973,A -85,B 0,C 180,E1 26765.724,E2 26765.724} C_VEL
LIN {X 0,Y 715.212,Z 1035.24,A -85,B 0,C 180,E1 26764.427,E2 26764.427} C_VEL
LIN {X 0,Y 714.593,Z 1056.131,A -85,B 0,C 180,E1 26762.785,E2 26762.785} C_VEL
LIN {X 0,Y 713.971,Z 1075.416,A -85,B 0,C 180,E1 26761.067,E2 26761.067} C_VEL
LIN {X 0,Y 713.518,Z 1091.702,A -85,B 0,C 180,E1 26759.463,E2 26759.463} C_VEL
LIN {X 0,Y 713.057,Z 1110.462,A -85,B 0,C 180,E1 26757.382,E2 26757.382} C_VEL
LIN {X 0,Y 712.729,Z 1124.012,A -85,B 0,C 180,E1 26755.689,E2 26755.689} C_VEL
LIN {X 0,Y 712.491,Z 1136.217,A -85,B 0,C 180,E1 26753.992,E2 26753.992} C_VEL
LIN {X 0,Y 712.29,Z 1149.602,A -85,B 0,C 180,E1 26751.891,E2 26751.891} C_VEL
LIN {X 0,Y 712.118,Z 1160.575,A -85,B 0,C 180,E1 26749.864,E2 26749.864} C_VEL
LIN {X 0,Y 712.015,Z 1168.576,A -85,B 0,C 180,E1 26748.164,E2 26748.164} C_VEL
LIN {X 0,Y 711.981,Z 1176.128,A -85,B 0,C 180,E1 26746.312,E2 26746.312} C_VEL
LIN {X 0,Y 711.937,Z 1183.25,A -85,B 0,C 180,E1 26744.144,E2 26744.144} C_VEL
LIN {X 0,Y 711.916,Z 1188.604,A -85,B 0,C 180,E1 26741.997,E2 26741.997} C_VEL
LIN {X 0,Y 711.908,Z 1192.321,A -85,B 0,C 180,E1 26739.866,E2 26739.866} C_VEL
LIN {X 0,Y 711.905,Z 1194.478,A -85,B 0,C 180,E1 26737.667,E2 26737.667} C_VEL
LIN {X 0,Y 711.893,Z 1194.874,A -85,B 0,C 180,E1 26735.48,E2 26735.48} C_VEL
LIN {X 0,Y 711.907,Z 1193.97,A -85,B 0,C 180,E1 26733.543,E2 26733.543} C_VEL
LIN {X 0,Y 711.908,Z 1191.311,A -85,B 0,C 180,E1 26731.368,E2 26731.368} C_VEL
LIN {X 0,Y 711.919,Z 1187.187,A -85,B 0,C 180,E1 26729.275,E2 26729.275} C_VEL
LIN {X 0,Y 711.947,Z 1181.247,A -85,B 0,C 180,E1 26727.102,E2 26727.102} C_VEL
LIN {X 0,Y 711.995,Z 1173.559,A -85,B 0,C 180,E1 26724.924,E2 26724.924} C_VEL
LIN {X 0,Y 712.092,Z 1163.614,A -85,B 0,C 180,E1 26722.659,E2 26722.659} C_VEL
LIN {X 0,Y 712.183,Z 1154.365,A -85,B 0,C 180,E1 26720.871,E2 26720.871} C_VEL
LIN {X 0,Y 712.356,Z 1144.286,A -85,B 0,C 180,E1 26719.159,E2 26719.159} C_VEL
LIN {X 0,Y 712.586,Z 1132.333,A -85,B 0,C 180,E1 26717.356,E2 26717.356} C_VEL
LIN {X 0,Y 712.916,Z 1116.136,A -85,B 0,C 180,E1 26715.211,E2 26715.211} C_VEL
LIN {X 0,Y 713.259,Z 1101.176,A -85,B 0,C 180,E1 26713.466,E2 26713.466} C_VEL
LIN {X 0,Y 713.725,Z 1085.116,A -85,B 0,C 180,E1 26711.777,E2 26711.777} C_VEL
LIN {X 0,Y 714.263,Z 1065.064,A -85,B 0,C 180,E1 26709.899,E2 26709.899} C_VEL
LIN {X 0,Y 714.817,Z 1047.978,A -85,B 0,C 180,E1 26708.468,E2 26708.468} C_VEL
LIN {X 0,Y 715.441,Z 1028.798,A -85,B 0,C 180,E1 26707.007,E2 26707.007} C_VEL
LIN {X 0,Y 716.172,Z 1005.203,A -85,B 0,C 180,E1 26705.414,E2 26705.414} C_VEL
LIN {X 0,Y 716.826,Z 985.723,A -85,B 0,C 180,E1 26704.246,E2 26704.246} C_VEL
LIN {X 0,Y 717.499,Z 965.524,A -85,B 0,C 180,E1 26703.159,E2 26703.159} C_VEL
LIN {X 0,Y 718.326,Z 940.693,A -85,B 0,C 180,E1 26701.979,E2 26701.979} C_VEL
LIN {X 0,Y 718.965,Z 915.502,A -85,B 0,C 180,E1 26700.964,E2 26700.964} C_VEL
LIN {X 0,Y 719.515,Z 894.429,A -85,B 0,C 180,E1 26700.234,E2 26700.234} C_VEL
LIN {X 0,Y 720.108,Z 871.479,A -85,B 0,C 180,E1 26699.556,E2 26699.556} C_VEL
LIN {X 0,Y 720.668,Z 843.892,A -85,B 0,C 180,E1 26698.91,E2 26698.91} C_VEL
LIN {X 0,Y 721.046,Z 817.488,A -85,B 0,C 180,E1 26698.454,E2 26698.454} C_VEL
LIN {X 0,Y 722.498,Z 588.645,A -85,B 0,C 180,E1 26695.659,E2 26695.659} C_VEL
LIN {X 0,Y 723.904,Z 371.548,A -85,B 0,C 180,E1 26692.931,E2 26692.931} C_VEL
LIN {X 0,Y 723.885,Z 353.664,A -85,B 0,C 180,E1 26692.691,E2 26692.691} C_VEL
LIN {X 0,Y 721.231,Z 344.541,A -85,B 0,C 180,E1 26692.37,E2 26692.37} C_VEL
LIN {X 0,Y 718.839,Z 340.708,A -85,B 0,C 180,E1 26692.128,E2 26692.128} C_VEL
LIN {X 0,Y 713.378,Z 328.697,A -85,B 0,C 180,E1 26690.814,E2 26690.814} C_VEL
LIN {X 0,Y 712.252,Z 325.512,A -85,B 0,C 180,E1 26690.469,E2 26690.469} C_VEL
LIN {X 0,Y 712.273,Z 325.501,A -85,B 0,C 180,E1 26687.596,E2 26687.596} C_VEL
LIN {X 0,Y 712.256,Z 325.511,A -85,B 0,C 180,E1 26684.624,E2 26684.624} C_VEL
LIN {X 0,Y 712.28,Z 325.501,A -85,B 0,C 180,E1 26681.685,E2 26681.685} C_VEL
LIN {X 0,Y 712.265,Z 325.51,A -85,B 0,C 180,E1 26678.66,E2 26678.66} C_VEL
LIN {X 0,Y 712.257,Z 325.502,A -85,B 0,C 180,E1 26675.732,E2 26675.732} C_VEL
LIN {X 0,Y 712.268,Z 325.511,A -85,B 0,C 180,E1 26672.619,E2 26672.619} C_VEL
LIN {X 0,Y 712.236,Z 325.505,A -85,B 0,C 180,E1 26669.8,E2 26669.8} C_VEL
LIN {X 0,Y 712.278,Z 325.497,A -85,B 0,C 180,E1 26666.874,E2 26666.874} C_VEL
LIN {X 0,Y 712.229,Z 325.508,A -85,B 0,C 180,E1 26664.025,E2 26664.025} C_VEL
LIN {X 0,Y 712.263,Z 325.497,A -85,B 0,C 180,E1 26661.231,E2 26661.231} C_VEL
LIN {X 0,Y 712.239,Z 325.51,A -85,B 0,C 180,E1 26658.159,E2 26658.159} C_VEL
LIN {X 0,Y 712.223,Z 325.502,A -85,B 0,C 180,E1 26655.471,E2 26655.471} C_VEL
LIN {X 0,Y 712.282,Z 325.493,A -85,B 0,C 180,E1 26652.567,E2 26652.567} C_VEL
LIN {X 0,Y 712.213,Z 325.507,A -85,B 0,C 180,E1 26649.699,E2 26649.699} C_VEL
LIN {X 0,Y 712.227,Z 325.506,A -85,B 0,C 180,E1 26647.097,E2 26647.097} C_VEL
LIN {X 0,Y 712.242,Z 325.511,A -85,B 0,C 180,E1 26644.025,E2 26644.025} C_VEL
LIN {X 0,Y 712.201,Z 325.506,A -85,B 0,C 180,E1 26641.448,E2 26641.448} C_VEL
LIN {X 0,Y 712.214,Z 325.507,A -85,B 0,C 180,E1 26638.954,E2 26638.954} C_VEL
LIN {X 0,Y 712.238,Z 325.51,A -85,B 0,C 180,E1 26635.894,E2 26635.894} C_VEL
LIN {X 0,Y 712.193,Z 325.51,A -85,B 0,C 180,E1 26633.308,E2 26633.308} C_VEL
LIN {X 0,Y 712.192,Z 325.507,A -85,B 0,C 180,E1 26630.953,E2 26630.953} C_VEL
LIN {X 0,Y 712.279,Z 325.504,A -85,B 0,C 180,E1 26628.091,E2 26628.091} C_VEL
LIN {X 0,Y 712.187,Z 325.507,A -85,B 0,C 180,E1 26625.279,E2 26625.279} C_VEL
LIN {X 0,Y 712.178,Z 325.512,A -85,B 0,C 180,E1 26622.936,E2 26622.936} C_VEL
LIN {X 0,Y 712.205,Z 325.502,A -85,B 0,C 180,E1 26620.394,E2 26620.394} C_VEL
LIN {X 0,Y 712.191,Z 325.512,A -85,B 0,C 180,E1 26617.288,E2 26617.288} C_VEL
LIN {X 0,Y 712.168,Z 325.498,A -85,B 0,C 180,E1 26614.823,E2 26614.823} C_VEL
LIN {X 0,Y 712.188,Z 325.512,A -85,B 0,C 180,E1 26612.399,E2 26612.399} C_VEL
LIN {X 0,Y 712.244,Z 325.508,A -85,B 0,C 180,E1 26609.456,E2 26609.456} C_VEL
LIN {X 0,Y 712.185,Z 325.512,A -85,B 0,C 180,E1 26606.8,E2 26606.8} C_VEL
LIN {X 0,Y 712.191,Z 325.513,A -85,B 0,C 180,E1 26604.363,E2 26604.363} C_VEL
LIN {X 0,Y 712.284,Z 325.511,A -85,B 0,C 180,E1 26601.547,E2 26601.547} C_VEL
LIN {X 0,Y 712.198,Z 325.512,A -85,B 0,C 180,E1 26598.686,E2 26598.686} C_VEL
LIN {X 0,Y 712.205,Z 325.544,A -85,B 0,C 180,E1 26596.182,E2 26596.182} C_VEL
LIN {X 0,Y 713.382,Z 328.762,A -85,B 0,C 180,E1 26595.844,E2 26595.844} C_VEL
LIN {X 0,Y 716.199,Z 334.795,A -85,B 0,C 180,E1 26595.171,E2 26595.171} C_VEL
LIN {X 0,Y 720.623,Z 344.747,A -85,B 0,C 180,E1 26594.106,E2 26594.106} C_VEL
LIN {X 0,Y 720.619,Z 351.282,A -85,B 0,C 180,E1 26593.676,E2 26593.676} C_VEL
LIN {X 0,Y 724.01,Z 364.314,A -85,B 0,C 180,E1 26593.246,E2 26593.246} C_VEL
LIN {X 0,Y 722.646,Z 574.749,A -85,B 0,C 180,E1 26590.592,E2 26590.592} C_VEL
LIN {X 0,Y 721.298,Z 799.019,A -85,B 0,C 180,E1 26587.858,E2 26587.858} C_VEL
LIN {X 0,Y 720.974,Z 835.225,A -85,B 0,C 180,E1 26587.385,E2 26587.385} C_VEL
LIN {X 0,Y 720.481,Z 862.662,A -85,B 0,C 180,E1 26586.858,E2 26586.858} C_VEL
LIN {X 0,Y 719.968,Z 888.091,A -85,B 0,C 180,E1 26586.218,E2 26586.218} C_VEL
LIN {X 0,Y 719.285,Z 916.179,A -85,B 0,C 180,E1 26585.33,E2 26585.33} C_VEL
LIN {X 0,Y 718.6,Z 939.477,A -85,B 0,C 180,E1 26584.445,E2 26584.445} C_VEL
LIN {X 0,Y 717.941,Z 960.685,A -85,B 0,C 180,E1 26583.519,E2 26583.519} C_VEL
LIN {X 0,Y 717.251,Z 982.975,A -85,B 0,C 180,E1 26582.413,E2 26582.413} C_VEL
LIN {X 0,Y 716.465,Z 1007.878,A -85,B 0,C 180,E1 26580.995,E2 26580.995} C_VEL
LIN {X 0,Y 715.787,Z 1027.564,A -85,B 0,C 180,E1 26579.729,E2 26579.729} C_VEL
LIN {X 0,Y 715.19,Z 1045.813,A -85,B 0,C 180,E1 26578.431,E2 26578.431} C_VEL
LIN {X 0,Y 714.548,Z 1067.21,A -85,B 0,C 180,E1 26576.736,E2 26576.736} C_VEL
LIN {X 0,Y 713.971,Z 1085.445,A -85,B 0,C 180,E1 26575.109,E2 26575.109} C_VEL
LIN {X 0,Y 713.51,Z 1101.39,A -85,B 0,C 180,E1 26573.54,E2 26573.54} C_VEL
LIN {X 0,Y 713.048,Z 1120.122,A -85,B 0,C 180,E1 26571.469,E2 26571.469} C_VEL
LIN {X 0,Y 712.742,Z 1134.091,A -85,B 0,C 180,E1 26569.723,E2 26569.723} C_VEL
LIN {X 0,Y 712.498,Z 1146.001,A -85,B 0,C 180,E1 26568.068,E2 26568.068} C_VEL
LIN {X 0,Y 712.28,Z 1158.897,A -85,B 0,C 180,E1 26566.054,E2 26566.054} C_VEL
LIN {X 0,Y 712.123,Z 1170.242,A -85,B 0,C 180,E1 26563.975,E2 26563.975} C_VEL
LIN {X 0,Y 712.027,Z 1178.431,A -85,B 0,C 180,E1 26562.242,E2 26562.242} C_VEL
LIN {X 0,Y 711.98,Z 1186.132,A -85,B 0,C 180,E1 26560.356,E2 26560.356} C_VEL
LIN {X 0,Y 711.936,Z 1193.353,A -85,B 0,C 180,E1 26558.155,E2 26558.155} C_VEL
LIN {X 0,Y 711.917,Z 1198.764,A -85,B 0,C 180,E1 26555.966,E2 26555.966} C_VEL
LIN {X 0,Y 711.907,Z 1202.381,A -85,B 0,C 180,E1 26553.866,E2 26553.866} C_VEL
LIN {X 0,Y 711.909,Z 1204.549,A -85,B 0,C 180,E1 26551.61,E2 26551.61} C_VEL
LIN {X 0,Y 711.89,Z 1204.872,A -85,B 0,C 180,E1 26549.517,E2 26549.517} C_VEL
LIN {X 0,Y 711.907,Z 1203.967,A -85,B 0,C 180,E1 26547.585,E2 26547.585} C_VEL
LIN {X 0,Y 711.908,Z 1201.304,A -85,B 0,C 180,E1 26545.409,E2 26545.409} C_VEL
LIN {X 0,Y 711.918,Z 1197.153,A -85,B 0,C 180,E1 26543.306,E2 26543.306} C_VEL
LIN {X 0,Y 711.945,Z 1191.397,A -85,B 0,C 180,E1 26541.195,E2 26541.195} C_VEL
LIN {X 0,Y 711.977,Z 1183.958,A -85,B 0,C 180,E1 26539.072,E2 26539.072} C_VEL
LIN {X 0,Y 712.09,Z 1173.94,A -85,B 0,C 180,E1 26536.77,E2 26536.77} C_VEL
LIN {X 0,Y 712.178,Z 1164.532,A -85,B 0,C 180,E1 26534.946,E2 26534.946} C_VEL
LIN {X 0,Y 712.341,Z 1154.745,A -85,B 0,C 180,E1 26533.277,E2 26533.277} C_VEL
LIN {X 0,Y 712.542,Z 1143.678,A -85,B 0,C 180,E1 26531.595,E2 26531.595} C_VEL
LIN {X 0,Y 712.858,Z 1129.296,A -85,B 0,C 180,E1 26529.644,E2 26529.644} C_VEL
LIN {X 0,Y 713.224,Z 1112.624,A -85,B 0,C 180,E1 26527.672,E2 26527.672} C_VEL
LIN {X 0,Y 713.611,Z 1097.982,A -85,B 0,C 180,E1 26526.114,E2 26526.114} C_VEL
LIN {X 0,Y 714.174,Z 1079.332,A -85,B 0,C 180,E1 26524.317,E2 26524.317} C_VEL
LIN {X 0,Y 714.745,Z 1059.885,A -85,B 0,C 180,E1 26522.665,E2 26522.665} C_VEL
LIN {X 0,Y 715.326,Z 1042.237,A -85,B 0,C 180,E1 26521.306,E2 26521.306} C_VEL
LIN {X 0,Y 716.075,Z 1020.247,A -85,B 0,C 180,E1 26519.777,E2 26519.777} C_VEL
LIN {X 0,Y 716.773,Z 997.041,A -85,B 0,C 180,E1 26518.365,E2 26518.365} C_VEL
LIN {X 0,Y 717.452,Z 976.757,A -85,B 0,C 180,E1 26517.267,E2 26517.267} C_VEL
LIN {X 0,Y 718.191,Z 954.379,A -85,B 0,C 180,E1 26516.192,E2 26516.192} C_VEL
LIN {X 0,Y 718.939,Z 927.681,A -85,B 0,C 180,E1 26515.09,E2 26515.09} C_VEL
LIN {X 0,Y 719.504,Z 905.589,A -85,B 0,C 180,E1 26514.316,E2 26514.316} C_VEL
LIN {X 0,Y 720.071,Z 882.536,A -85,B 0,C 180,E1 26513.63,E2 26513.63} C_VEL
LIN {X 0,Y 720.646,Z 855.582,A -85,B 0,C 180,E1 26512.989,E2 26512.989} C_VEL
LIN {X 0,Y 721.042,Z 828.374,A -85,B 0,C 180,E1 26512.511,E2 26512.511} C_VEL
LIN {X 0,Y 722.49,Z 599.203,A -85,B 0,C 180,E1 26509.71,E2 26509.71} C_VEL
LIN {X 0,Y 723.792,Z 395.098,A -85,B 0,C 180,E1 26507.147,E2 26507.147} C_VEL
LIN {X 0,Y 723.842,Z 363.088,A -85,B 0,C 180,E1 26506.725,E2 26506.725} C_VEL
LIN {X 0,Y 720.488,Z 350.368,A -85,B 0,C 180,E1 26506.282,E2 26506.282} C_VEL
LIN {X 0,Y 720.46,Z 344.144,A -85,B 0,C 180,E1 26505.839,E2 26505.839} C_VEL
LIN {X 0,Y 713.804,Z 329.357,A -85,B 0,C 180,E1 26504.235,E2 26504.235} C_VEL
LIN {X 0,Y 712.256,Z 325.863,A -85,B 0,C 180,E1 26503.846,E2 26503.846} C_VEL
LIN {X 0,Y 712.203,Z 325.517,A -85,B 0,C 180,E1 26503.8,E2 26503.8} C_VEL
LIN {X 0,Y 712.201,Z 325.514,A -85,B 0,C 180,E1 26501.289,E2 26501.289} C_VEL
LIN {X 0,Y 712.282,Z 325.51,A -85,B 0,C 180,E1 26498.437,E2 26498.437} C_VEL
LIN {X 0,Y 712.194,Z 325.51,A -85,B 0,C 180,E1 26495.623,E2 26495.623} C_VEL
LIN {X 0,Y 712.189,Z 325.51,A -85,B 0,C 180,E1 26493.199,E2 26493.199} C_VEL
LIN {X 0,Y 712.257,Z 325.5,A -85,B 0,C 180,E1 26490.466,E2 26490.466} C_VEL
LIN {X 0,Y 712.197,Z 325.508,A -85,B 0,C 180,E1 26487.601,E2 26487.601} C_VEL
LIN {X 0,Y 712.178,Z 325.509,A -85,B 0,C 180,E1 26485.177,E2 26485.177} C_VEL
LIN {X 0,Y 712.186,Z 325.51,A -85,B 0,C 180,E1 26482.799,E2 26482.799} C_VEL
LIN {X 0,Y 712.265,Z 325.509,A -85,B 0,C 180,E1 26479.946,E2 26479.946} C_VEL
LIN {X 0,Y 712.172,Z 325.503,A -85,B 0,C 180,E1 26477.148,E2 26477.148} C_VEL
LIN {X 0,Y 712.17,Z 325.511,A -85,B 0,C 180,E1 26474.805,E2 26474.805} C_VEL
LIN {X 0,Y 712.214,Z 325.511,A -85,B 0,C 180,E1 26472.239,E2 26472.239} C_VEL
LIN {X 0,Y 712.192,Z 325.512,A -85,B 0,C 180,E1 26469.21,E2 26469.21} C_VEL
LIN {X 0,Y 712.176,Z 325.506,A -85,B 0,C 180,E1 26466.773,E2 26466.773} C_VEL
LIN {X 0,Y 712.19,Z 325.507,A -85,B 0,C 180,E1 26464.348,E2 26464.348} C_VEL
LIN {X 0,Y 712.262,Z 325.499,A -85,B 0,C 180,E1 26461.448,E2 26461.448} C_VEL
LIN {X 0,Y 712.189,Z 325.508,A -85,B 0,C 180,E1 26458.713,E2 26458.713} C_VEL
LIN {X 0,Y 712.189,Z 325.51,A -85,B 0,C 180,E1 26456.297,E2 26456.297} C_VEL
LIN {X 0,Y 712.28,Z 325.502,A -85,B 0,C 180,E1 26453.471,E2 26453.471} C_VEL
LIN {X 0,Y 712.201,Z 325.504,A -85,B 0,C 180,E1 26450.627,E2 26450.627} C_VEL
LIN {X 0,Y 712.196,Z 325.505,A -85,B 0,C 180,E1 26448.172,E2 26448.172} C_VEL
LIN {X 0,Y 712.264,Z 325.504,A -85,B 0,C 180,E1 26445.446,E2 26445.446} C_VEL
LIN {X 0,Y 712.215,Z 325.508,A -85,B 0,C 180,E1 26442.516,E2 26442.516} C_VEL
LIN {X 0,Y 712.267,Z 325.5,A -85,B 0,C 180,E1 26440.904,E2 26440.904} C_VEL
LIN {X 0,Y 711.225,Z 325.624,A -85,B 0,C 180,E1 26440.284,E2 26440.284} C_VEL
LIN {X 0,Y 704.795,Z 326.434,A -85,B 0,C 180,E1 26438.548,E2 26438.548} C_VEL
LIN {X 0,Y 704.265,Z 326.497,A -85,B 0,C 180,E1 26438.097,E2 26438.097} C_VEL
LIN {X 0,Y 704.302,Z 326.491,A -85,B 0,C 180,E1 26435.419,E2 26435.419} C_VEL
LIN {X 0,Y 704.29,Z 326.495,A -85,B 0,C 180,E1 26432.338,E2 26432.338} C_VEL
LIN {X 0,Y 704.274,Z 326.497,A -85,B 0,C 180,E1 26429.734,E2 26429.734} C_VEL
LIN {X 0,Y 704.344,Z 326.499,A -85,B 0,C 180,E1 26426.869,E2 26426.869} C_VEL
LIN {X 0,Y 704.283,Z 326.501,A -85,B 0,C 180,E1 26423.9,E2 26423.9} C_VEL
LIN {X 0,Y 704.303,Z 326.588,A -85,B 0,C 180,E1 26422.004,E2 26422.004} C_VEL
LIN {X 0,Y 705.599,Z 330.006,A -85,B 0,C 180,E1 26421.634,E2 26421.634} C_VEL
LIN {X 0,Y 710.74,Z 341.251,A -85,B 0,C 180,E1 26420.396,E2 26420.396} C_VEL
LIN {X 0,Y 716.44,Z 350.086,A -85,B 0,C 180,E1 26419.831,E2 26419.831} C_VEL
LIN {X 0,Y 718.176,Z 357.341,A -85,B 0,C 180,E1 26419.599,E2 26419.599} C_VEL
LIN {X 0,Y 716.497,Z 574.199,A -85,B 0,C 180,E1 26416.847,E2 26416.847} C_VEL
LIN {X 0,Y 714.887,Z 801.467,A -85,B 0,C 180,E1 26414.058,E2 26414.058} C_VEL
LIN {X 0,Y 714.476,Z 831.067,A -85,B 0,C 180,E1 26413.632,E2 26413.632} C_VEL
LIN {X 0,Y 713.936,Z 856.678,A -85,B 0,C 180,E1 26413.11,E2 26413.11} C_VEL
LIN {X 0,Y 713.275,Z 883.605,A -85,B 0,C 180,E1 26412.4,E2 26412.4} C_VEL
LIN {X 0,Y 712.479,Z 909.742,A -85,B 0,C 180,E1 26411.536,E2 26411.536} C_VEL
LIN {X 0,Y 711.789,Z 930.541,A -85,B 0,C 180,E1 26410.73,E2 26410.73} C_VEL
LIN {X 0,Y 711.075,Z 950.575,A -85,B 0,C 180,E1 26409.846,E2 26409.846} C_VEL
LIN {X 0,Y 710.313,Z 970.77,A -85,B 0,C 180,E1 26408.842,E2 26408.842} C_VEL
LIN {X 0,Y 709.427,Z 995.257,A -85,B 0,C 180,E1 26407.461,E2 26407.461} C_VEL
LIN {X 0,Y 708.574,Z 1016.455,A -85,B 0,C 180,E1 26406.095,E2 26406.095} C_VEL
LIN {X 0,Y 707.868,Z 1034.645,A -85,B 0,C 180,E1 26404.796,E2 26404.796} C_VEL
LIN {X 0,Y 707.102,Z 1055.329,A -85,B 0,C 180,E1 26403.161,E2 26403.161} C_VEL
LIN {X 0,Y 706.402,Z 1075.043,A -85,B 0,C 180,E1 26401.391,E2 26401.391} C_VEL
LIN {X 0,Y 705.86,Z 1090.924,A -85,B 0,C 180,E1 26399.815,E2 26399.815} C_VEL
LIN {X 0,Y 705.326,Z 1109.101,A -85,B 0,C 180,E1 26397.797,E2 26397.797} C_VEL
LIN {X 0,Y 704.9,Z 1123.916,A -85,B 0,C 180,E1 26395.931,E2 26395.931} C_VEL
LIN {X 0,Y 704.614,Z 1136.151,A -85,B 0,C 180,E1 26394.211,E2 26394.211} C_VEL
LIN {X 0,Y 704.354,Z 1149.48,A -85,B 0,C 180,E1 26392.097,E2 26392.097} C_VEL
LIN {X 0,Y 704.159,Z 1160.64,A -85,B 0,C 180,E1 26390.011,E2 26390.011} C_VEL
LIN {X 0,Y 704.046,Z 1168.634,A -85,B 0,C 180,E1 26388.292,E2 26388.292} C_VEL
LIN {X 0,Y 703.996,Z 1176.174,A -85,B 0,C 180,E1 26386.417,E2 26386.417} C_VEL
LIN {X 0,Y 703.943,Z 1183.29,A -85,B 0,C 180,E1 26384.224,E2 26384.224} C_VEL
LIN {X 0,Y 703.917,Z 1188.632,A -85,B 0,C 180,E1 26382.052,E2 26382.052} C_VEL
LIN {X 0,Y 703.908,Z 1192.338,A -85,B 0,C 180,E1 26379.897,E2 26379.897} C_VEL
LIN {X 0,Y 703.906,Z 1194.487,A -85,B 0,C 180,E1 26377.673,E2 26377.673} C_VEL
LIN {X 0,Y 703.894,Z 1194.87,A -85,B 0,C 180,E1 26375.461,E2 26375.461} C_VEL
LIN {X 0,Y 703.906,Z 1193.955,A -85,B 0,C 180,E1 26373.501,E2 26373.501} C_VEL
LIN {X 0,Y 703.909,Z 1191.29,A -85,B 0,C 180,E1 26371.302,E2 26371.302} C_VEL
LIN {X 0,Y 703.921,Z 1187.155,A -85,B 0,C 180,E1 26369.186,E2 26369.186} C_VEL
LIN {X 0,Y 703.954,Z 1181.203,A -85,B 0,C 180,E1 26366.987,E2 26366.987} C_VEL
LIN {X 0,Y 704.022,Z 1173.51,A -85,B 0,C 180,E1 26364.785,E2 26364.785} C_VEL
LIN {X 0,Y 704.122,Z 1163.555,A -85,B 0,C 180,E1 26362.493,E2 26362.493} C_VEL
LIN {X 0,Y 704.255,Z 1154.185,A -85,B 0,C 180,E1 26360.664,E2 26360.664} C_VEL
LIN {X 0,Y 704.453,Z 1144.215,A -85,B 0,C 180,E1 26358.953,E2 26358.953} C_VEL
LIN {X 0,Y 704.718,Z 1132.053,A -85,B 0,C 180,E1 26357.099,E2 26357.099} C_VEL
LIN {X 0,Y 705.109,Z 1115.985,A -85,B 0,C 180,E1 26354.952,E2 26354.952} C_VEL
LIN {X 0,Y 705.513,Z 1101.833,A -85,B 0,C 180,E1 26353.28,E2 26353.28} C_VEL
LIN {X 0,Y 706.04,Z 1086.012,A -85,B 0,C 180,E1 26351.59,E2 26351.59} C_VEL
LIN {X 0,Y 706.727,Z 1065.425,A -85,B 0,C 180,E1 26349.632,E2 26349.632} C_VEL
LIN {X 0,Y 707.359,Z 1048.248,A -85,B 0,C 180,E1 26348.176,E2 26348.176} C_VEL
LIN {X 0,Y 708.038,Z 1030.385,A -85,B 0,C 180,E1 26346.796,E2 26346.796} C_VEL
LIN {X 0,Y 708.943,Z 1006.406,A -85,B 0,C 180,E1 26345.147,E2 26345.147} C_VEL
LIN {X 0,Y 709.738,Z 986.279,A -85,B 0,C 180,E1 26343.925,E2 26343.925} C_VEL
LIN {X 0,Y 710.477,Z 966.981,A -85,B 0,C 180,E1 26342.872,E2 26342.872} C_VEL
LIN {X 0,Y 711.266,Z 946.16,A -85,B 0,C 180,E1 26341.859,E2 26341.859} C_VEL
LIN {X 0,Y 712.168,Z 919.939,A -85,B 0,C 180,E1 26340.752,E2 26340.752} C_VEL
LIN {X 0,Y 712.857,Z 896.218,A -85,B 0,C 180,E1 26339.909,E2 26339.909} C_VEL
LIN {X 0,Y 713.525,Z 873.497,A -85,B 0,C 180,E1 26339.224,E2 26339.224} C_VEL
LIN {X 0,Y 714.199,Z 846.317,A -85,B 0,C 180,E1 26338.57,E2 26338.57} C_VEL
LIN {X 0,Y 714.653,Z 819.565,A -85,B 0,C 180,E1 26338.092,E2 26338.092} C_VEL
LIN {X 0,Y 715.758,Z 675.395,A -85,B 0,C 180,E1 26336.316,E2 26336.316} C_VEL
LIN {X 0,Y 717.374,Z 457.556,A -85,B 0,C 180,E1 26333.594,E2 26333.594} C_VEL
LIN {X 0,Y 718.015,Z 355.818,A -85,B 0,C 180,E1 26332.278,E2 26332.278} C_VEL
LIN {X 0,Y 716.06,Z 349.291,A -85,B 0,C 180,E1 26332.039,E2 26332.039} C_VEL
LIN {X 0,Y 710.51,Z 340.79,A -85,B 0,C 180,E1 26331.486,E2 26331.486} C_VEL
LIN {X 0,Y 705.629,Z 329.991,A -85,B 0,C 180,E1 26330.277,E2 26330.277} C_VEL
LIN {X 0,Y 704.346,Z 326.495,A -85,B 0,C 180,E1 26329.872,E2 26329.872} C_VEL
LIN {X 0,Y 704.33,Z 326.501,A -85,B 0,C 180,E1 26326.823,E2 26326.823} C_VEL
LIN {X 0,Y 704.332,Z 326.492,A -85,B 0,C 180,E1 26323.849,E2 26323.849} C_VEL
LIN {X 0,Y 704.328,Z 326.5,A -85,B 0,C 180,E1 26320.705,E2 26320.705} C_VEL
LIN {X 0,Y 704.326,Z 326.49,A -85,B 0,C 180,E1 26317.725,E2 26317.725} C_VEL
LIN {X 0,Y 704.324,Z 326.5,A -85,B 0,C 180,E1 26314.575,E2 26314.575} C_VEL
LIN {X 0,Y 704.313,Z 326.493,A -85,B 0,C 180,E1 26311.687,E2 26311.687} C_VEL
LIN {X 0,Y 704.332,Z 326.495,A -85,B 0,C 180,E1 26308.582,E2 26308.582} C_VEL
LIN {X 0,Y 704.294,Z 326.484,A -85,B 0,C 180,E1 26305.749,E2 26305.749} C_VEL
LIN {X 0,Y 704.343,Z 326.497,A -85,B 0,C 180,E1 26302.802,E2 26302.802} C_VEL
LIN {X 0,Y 704.285,Z 326.486,A -85,B 0,C 180,E1 26299.974,E2 26299.974} C_VEL
LIN {X 0,Y 704.308,Z 326.493,A -85,B 0,C 180,E1 26297.26,E2 26297.26} C_VEL
LIN {X 0,Y 704.299,Z 326.48,A -85,B 0,C 180,E1 26294.134,E2 26294.134} C_VEL
LIN {X 0,Y 704.276,Z 326.494,A -85,B 0,C 180,E1 26291.465,E2 26291.465} C_VEL
LIN {X 0,Y 704.345,Z 326.494,A -85,B 0,C 180,E1 26288.572,E2 26288.572} C_VEL
LIN {X 0,Y 704.272,Z 326.495,A -85,B 0,C 180,E1 26285.704,E2 26285.704} C_VEL
LIN {X 0,Y 704.272,Z 326.497,A -85,B 0,C 180,E1 26283.174,E2 26283.174} C_VEL
LIN {X 0,Y 704.341,Z 326.498,A -85,B 0,C 180,E1 26280.244,E2 26280.244} C_VEL
LIN {X 0,Y 704.261,Z 326.498,A -85,B 0,C 180,E1 26277.477,E2 26277.477} C_VEL
LIN {X 0,Y 704.26,Z 326.496,A -85,B 0,C 180,E1 26275.032,E2 26275.032} C_VEL
LIN {X 0,Y 704.346,Z 326.497,A -85,B 0,C 180,E1 26272.167,E2 26272.167} C_VEL
LIN {X 0,Y 704.254,Z 326.5,A -85,B 0,C 180,E1 26269.364,E2 26269.364} C_VEL
LIN {X 0,Y 704.244,Z 326.488,A -85,B 0,C 180,E1 26266.953,E2 26266.953} C_VEL
LIN {X 0,Y 704.29,Z 326.494,A -85,B 0,C 180,E1 26264.351,E2 26264.351} C_VEL
LIN {X 0,Y 704.257,Z 326.49,A -85,B 0,C 180,E1 26261.37,E2 26261.37} C_VEL
LIN {X 0,Y 704.234,Z 326.497,A -85,B 0,C 180,E1 26258.878,E2 26258.878} C_VEL
LIN {X 0,Y 704.246,Z 326.501,A -85,B 0,C 180,E1 26256.486,E2 26256.486} C_VEL
LIN {X 0,Y 704.296,Z 326.498,A -85,B 0,C 180,E1 26253.526,E2 26253.526} C_VEL
LIN {X 0,Y 704.238,Z 326.5,A -85,B 0,C 180,E1 26250.856,E2 26250.856} C_VEL
LIN {X 0,Y 704.244,Z 326.498,A -85,B 0,C 180,E1 26248.5,E2 26248.5} C_VEL
LIN {X 0,Y 704.332,Z 326.5,A -85,B 0,C 180,E1 26245.695,E2 26245.695} C_VEL
LIN {X 0,Y 704.255,Z 326.502,A -85,B 0,C 180,E1 26242.783,E2 26242.783} C_VEL
LIN {X 0,Y 704.253,Z 326.506,A -85,B 0,C 180,E1 26240.395,E2 26240.395} C_VEL
LIN {X 0,Y 704.314,Z 326.499,A -85,B 0,C 180,E1 26237.701,E2 26237.701} C_VEL
LIN {X 0,Y 704.284,Z 326.603,A -85,B 0,C 180,E1 26236.777,E2 26236.777} C_VEL
LIN {X 0,Y 705.658,Z 330.127,A -85,B 0,C 180,E1 26236.391,E2 26236.391} C_VEL
LIN {X 0,Y 711.699,Z 343.19,A -85,B 0,C 180,E1 26234.92,E2 26234.92} C_VEL
LIN {X 0,Y 714.113,Z 348.878,A -85,B 0,C 180,E1 26234.316,E2 26234.316} C_VEL
LIN {X 0,Y 714.219,Z 351.372,A -85,B 0,C 180,E1 26234.167,E2 26234.167} C_VEL
LIN {X 0,Y 718.152,Z 366.514,A -85,B 0,C 180,E1 26233.657,E2 26233.657} C_VEL
LIN {X 0,Y 716.55,Z 576.35,A -85,B 0,C 180,E1 26230.99,E2 26230.99} C_VEL
LIN {X 0,Y 714.966,Z 800.291,A -85,B 0,C 180,E1 26228.238,E2 26228.238} C_VEL
LIN {X 0,Y 714.588,Z 835.553,A -85,B 0,C 180,E1 26227.771,E2 26227.771} C_VEL
LIN {X 0,Y 714.018,Z 862.838,A -85,B 0,C 180,E1 26227.243,E2 26227.243} C_VEL
LIN {X 0,Y 713.425,Z 888.088,A -85,B 0,C 180,E1 26226.604,E2 26226.604} C_VEL
LIN {X 0,Y 712.627,Z 916.176,A -85,B 0,C 180,E1 26225.71,E2 26225.71} C_VEL
LIN {X 0,Y 711.839,Z 939.48,A -85,B 0,C 180,E1 26224.819,E2 26224.819} C_VEL
LIN {X 0,Y 711.071,Z 960.688,A -85,B 0,C 180,E1 26223.886,E2 26223.886} C_VEL
LIN {X 0,Y 710.256,Z 982.229,A -85,B 0,C 180,E1 26222.812,E2 26222.812} C_VEL
LIN {X 0,Y 709.317,Z 1007.875,A -85,B 0,C 180,E1 26221.343,E2 26221.343} C_VEL
LIN {X 0,Y 708.532,Z 1027.566,A -85,B 0,C 180,E1 26220.065,E2 26220.065} C_VEL
LIN {X 0,Y 707.831,Z 1045.859,A -85,B 0,C 180,E1 26218.75,E2 26218.75} C_VEL
LIN {X 0,Y 707.057,Z 1066.703,A -85,B 0,C 180,E1 26217.088,E2 26217.088} C_VEL
LIN {X 0,Y 706.388,Z 1085.446,A -85,B 0,C 180,E1 26215.397,E2 26215.397} C_VEL
LIN {X 0,Y 705.819,Z 1101.773,A -85,B 0,C 180,E1 26213.773,E2 26213.773} C_VEL
LIN {X 0,Y 705.277,Z 1120.124,A -85,B 0,C 180,E1 26211.717,E2 26211.717} C_VEL
LIN {X 0,Y 704.919,Z 1133.806,A -85,B 0,C 180,E1 26209.989,E2 26209.989} C_VEL
LIN {X 0,Y 704.621,Z 1146.003,A -85,B 0,C 180,E1 26208.277,E2 26208.277} C_VEL
LIN {X 0,Y 704.353,Z 1158.896,A -85,B 0,C 180,E1 26206.24,E2 26206.24} C_VEL
LIN {X 0,Y 704.171,Z 1170.378,A -85,B 0,C 180,E1 26204.109,E2 26204.109} C_VEL
LIN {X 0,Y 704.062,Z 1178.432,A -85,B 0,C 180,E1 26202.383,E2 26202.383} C_VEL
LIN {X 0,Y 703.989,Z 1186.13,A -85,B 0,C 180,E1 26200.475,E2 26200.475} C_VEL
LIN {X 0,Y 703.943,Z 1193.353,A -85,B 0,C 180,E1 26198.248,E2 26198.248} C_VEL
LIN {X 0,Y 703.92,Z 1198.765,A -85,B 0,C 180,E1 26196.034,E2 26196.034} C_VEL
LIN {X 0,Y 703.908,Z 1202.381,A -85,B 0,C 180,E1 26193.91,E2 26193.91} C_VEL
LIN {X 0,Y 703.908,Z 1204.549,A -85,B 0,C 180,E1 26191.628,E2 26191.628} C_VEL
LIN {X 0,Y 703.89,Z 1204.872,A -85,B 0,C 180,E1 26189.512,E2 26189.512} C_VEL
LIN {X 0,Y 703.907,Z 1203.965,A -85,B 0,C 180,E1 26187.558,E2 26187.558} C_VEL
LIN {X 0,Y 703.909,Z 1201.428,A -85,B 0,C 180,E1 26185.438,E2 26185.438} C_VEL
LIN {X 0,Y 703.921,Z 1197.348,A -85,B 0,C 180,E1 26183.312,E2 26183.312} C_VEL
LIN {X 0,Y 703.949,Z 1191.394,A -85,B 0,C 180,E1 26181.094,E2 26181.094} C_VEL
LIN {X 0,Y 703.992,Z 1184.277,A -85,B 0,C 180,E1 26179.029,E2 26179.029} C_VEL
LIN {X 0,Y 704.128,Z 1173.942,A -85,B 0,C 180,E1 26176.617,E2 26176.617} C_VEL
LIN {X 0,Y 704.237,Z 1164.533,A -85,B 0,C 180,E1 26174.772,E2 26174.772} C_VEL
LIN {X 0,Y 704.436,Z 1154.7,A -85,B 0,C 180,E1 26173.076,E2 26173.076} C_VEL
LIN {X 0,Y 704.667,Z 1143.68,A -85,B 0,C 180,E1 26171.382,E2 26171.382} C_VEL
LIN {X 0,Y 705.059,Z 1128.62,A -85,B 0,C 180,E1 26169.322,E2 26169.322} C_VEL
LIN {X 0,Y 705.487,Z 1112.626,A -85,B 0,C 180,E1 26167.414,E2 26167.414} C_VEL
LIN {X 0,Y 705.974,Z 1097.611,A -85,B 0,C 180,E1 26165.8,E2 26165.8} C_VEL
LIN {X 0,Y 706.607,Z 1078.76,A -85,B 0,C 180,E1 26163.97,E2 26163.97} C_VEL
LIN {X 0,Y 707.315,Z 1059.611,A -85,B 0,C 180,E1 26162.331,E2 26162.331} C_VEL
LIN {X 0,Y 707.956,Z 1042.843,A -85,B 0,C 180,E1 26161.025,E2 26161.025} C_VEL
LIN {X 0,Y 708.731,Z 1022.919,A -85,B 0,C 180,E1 26159.618,E2 26159.618} C_VEL
LIN {X 0,Y 709.633,Z 998.649,A -85,B 0,C 180,E1 26158.105,E2 26158.105} C_VEL
LIN {X 0,Y 710.413,Z 978.54,A -85,B 0,C 180,E1 26156.997,E2 26156.997} C_VEL
LIN {X 0,Y 711.154,Z 958.818,A -85,B 0,C 180,E1 26156.027,E2 26156.027} C_VEL
LIN {X 0,Y 711.945,Z 936.924,A -85,B 0,C 180,E1 26155.076,E2 26155.076} C_VEL
LIN {X 0,Y 712.79,Z 910.723,A -85,B 0,C 180,E1 26154.102,E2 26154.102} C_VEL
LIN {X 0,Y 713.473,Z 885.508,A -85,B 0,C 180,E1 26153.325,E2 26153.325} C_VEL
LIN {X 0,Y 714.092,Z 860.326,A -85,B 0,C 180,E1 26152.702,E2 26152.702} C_VEL
LIN {X 0,Y 714.619,Z 832.66,A -85,B 0,C 180,E1 26152.183,E2 26152.183} C_VEL
LIN {X 0,Y 715.071,Z 784.577,A -85,B 0,C 180,E1 26151.572,E2 26151.572} C_VEL
LIN {X 0,Y 716.679,Z 559.863,A -85,B 0,C 180,E1 26148.804,E2 26148.804} C_VEL
LIN {X 0,Y 718.157,Z 365.918,A -85,B 0,C 180,E1 26146.335,E2 26146.335} C_VEL
LIN {X 0,Y 714.07,Z 350.368,A -85,B 0,C 180,E1 26145.788,E2 26145.788} C_VEL
LIN {X 0,Y 714,Z 348.336,A -85,B 0,C 180,E1 26145.636,E2 26145.636} C_VEL
LIN {X 0,Y 707.478,Z 334.016,A -85,B 0,C 180,E1 26144.056,E2 26144.056} C_VEL
LIN {X 0,Y 704.353,Z 327.027,A -85,B 0,C 180,E1 26143.262,E2 26143.262} C_VEL
LIN {X 0,Y 704.276,Z 326.506,A -85,B 0,C 180,E1 26143.182,E2 26143.182} C_VEL
LIN {X 0,Y 704.291,Z 326.503,A -85,B 0,C 180,E1 26140.075,E2 26140.075} C_VEL
LIN {X 0,Y 704.252,Z 326.501,A -85,B 0,C 180,E1 26137.473,E2 26137.473} C_VEL
LIN {X 0,Y 704.266,Z 326.498,A -85,B 0,C 180,E1 26134.997,E2 26134.997} C_VEL
LIN {X 0,Y 704.296,Z 326.496,A -85,B 0,C 180,E1 26131.975,E2 26131.975} C_VEL
LIN {X 0,Y 704.246,Z 326.5,A -85,B 0,C 180,E1 26129.423,E2 26129.423} C_VEL
LIN {X 0,Y 704.243,Z 326.496,A -85,B 0,C 180,E1 26127.102,E2 26127.102} C_VEL
LIN {X 0,Y 704.299,Z 326.497,A -85,B 0,C 180,E1 26124.402,E2 26124.402} C_VEL
LIN {X 0,Y 704.255,Z 326.493,A -85,B 0,C 180,E1 26121.488,E2 26121.488} C_VEL
LIN {X 0,Y 704.236,Z 326.502,A -85,B 0,C 180,E1 26119.06,E2 26119.06} C_VEL
LIN {X 0,Y 704.245,Z 326.491,A -85,B 0,C 180,E1 26116.595,E2 26116.595} C_VEL
LIN {X 0,Y 704.293,Z 326.499,A -85,B 0,C 180,E1 26113.631,E2 26113.631} C_VEL
LIN {X 0,Y 704.235,Z 326.49,A -85,B 0,C 180,E1 26110.968,E2 26110.968} C_VEL
LIN {X 0,Y 704.238,Z 326.502,A -85,B 0,C 180,E1 26108.574,E2 26108.574} C_VEL
LIN {X 0,Y 704.328,Z 326.485,A -85,B 0,C 180,E1 26105.785,E2 26105.785} C_VEL
LIN {X 0,Y 704.252,Z 326.5,A -85,B 0,C 180,E1 26102.93,E2 26102.93} C_VEL
LIN {X 0,Y 704.244,Z 326.488,A -85,B 0,C 180,E1 26100.569,E2 26100.569} C_VEL
LIN {X 0,Y 704.263,Z 326.499,A -85,B 0,C 180,E1 26098.129,E2 26098.129} C_VEL
LIN {X 0,Y 704.295,Z 326.484,A -85,B 0,C 180,E1 26095.113,E2 26095.113} C_VEL
LIN {X 0,Y 704.253,Z 326.499,A -85,B 0,C 180,E1 26092.494,E2 26092.494} C_VEL
LIN {X 0,Y 704.264,Z 326.494,A -85,B 0,C 180,E1 26090.025,E2 26090.025} C_VEL
LIN {X 0,Y 704.324,Z 326.496,A -85,B 0,C 180,E1 26087.038,E2 26087.038} C_VEL
LIN {X 0,Y 704.26,Z 326.483,A -85,B 0,C 180,E1 26084.35,E2 26084.35} C_VEL
LIN {X 0,Y 704.269,Z 326.499,A -85,B 0,C 180,E1 26081.885,E2 26081.885} C_VEL
LIN {X 0,Y 704.345,Z 326.489,A -85,B 0,C 180,E1 26078.951,E2 26078.951} C_VEL
LIN {X 0,Y 704.265,Z 326.497,A -85,B 0,C 180,E1 26078.097,E2 26078.097} C_VEL
LIN {X 0,Y 703.268,Z 326.63,A -85,B 0,C 180,E1 26077.47,E2 26077.47} C_VEL
LIN {X 0,Y 696.868,Z 327.418,A -85,B 0,C 180,E1 26075.714,E2 26075.714} C_VEL
LIN {X 0,Y 696.384,Z 327.475,A -85,B 0,C 180,E1 26075.258,E2 26075.258} C_VEL
LIN {X 0,Y 696.346,Z 327.484,A -85,B 0,C 180,E1 26072.274,E2 26072.274} C_VEL
LIN {X 0,Y 696.339,Z 327.486,A -85,B 0,C 180,E1 26069.652,E2 26069.652} C_VEL
LIN {X 0,Y 696.408,Z 327.487,A -85,B 0,C 180,E1 26066.738,E2 26066.738} C_VEL
LIN {X 0,Y 696.341,Z 327.492,A -85,B 0,C 180,E1 26063.801,E2 26063.801} C_VEL
LIN {X 0,Y 696.418,Z 327.582,A -85,B 0,C 180,E1 26062.603,E2 26062.603} C_VEL
LIN {X 0,Y 697.533,Z 330.742,A -85,B 0,C 180,E1 26062.259,E2 26062.259} C_VEL
LIN {X 0,Y 702.443,Z 341.257,A -85,B 0,C 180,E1 26061.064,E2 26061.064} C_VEL
LIN {X 0,Y 711.303,Z 354.733,A -85,B 0,C 180,E1 26060.166,E2 26060.166} C_VEL
LIN {X 0,Y 712.356,Z 359.534,A -85,B 0,C 180,E1 26060.017,E2 26060.017} C_VEL
LIN {X 0,Y 710.422,Z 576.322,A -85,B 0,C 180,E1 26057.244,E2 26057.244} C_VEL
LIN {X 0,Y 708.565,Z 803.978,A -85,B 0,C 180,E1 26054.428,E2 26054.428} C_VEL
LIN {X 0,Y 708.08,Z 832.578,A -85,B 0,C 180,E1 26054.003,E2 26054.003} C_VEL
LIN {X 0,Y 707.475,Z 857.785,A -85,B 0,C 180,E1 26053.479,E2 26053.479} C_VEL
LIN {X 0,Y 706.73,Z 884.271,A -85,B 0,C 180,E1 26052.773,E2 26052.773} C_VEL
LIN {X 0,Y 705.83,Z 910.018,A -85,B 0,C 180,E1 26051.912,E2 26051.912} C_VEL
LIN {X 0,Y 705.039,Z 930.895,A -85,B 0,C 180,E1 26051.096,E2 26051.096} C_VEL
LIN {X 0,Y 704.256,Z 950.168,A -85,B 0,C 180,E1 26050.24,E2 26050.24} C_VEL
LIN {X 0,Y 703.372,Z 970.613,A -85,B 0,C 180,E1 26049.217,E2 26049.217} C_VEL
LIN {X 0,Y 702.331,Z 994.76,A -85,B 0,C 180,E1 26047.849,E2 26047.849} C_VEL
LIN {X 0,Y 701.337,Z 1016.64,A -85,B 0,C 180,E1 26046.426,E2 26046.426} C_VEL
LIN {X 0,Y 700.52,Z 1034.81,A -85,B 0,C 180,E1 26045.114,E2 26045.114} C_VEL
LIN {X 0,Y 699.636,Z 1055.287,A -85,B 0,C 180,E1 26043.48,E2 26043.48} C_VEL
LIN {X 0,Y 698.834,Z 1074.922,A -85,B 0,C 180,E1 26041.699,E2 26041.699} C_VEL
LIN {X 0,Y 698.197,Z 1091.043,A -85,B 0,C 180,E1 26040.081,E2 26040.081} C_VEL
LIN {X 0,Y 697.549,Z 1109.581,A -85,B 0,C 180,E1 26037.994,E2 26037.994} C_VEL
LIN {X 0,Y 697.075,Z 1124.2,A -85,B 0,C 180,E1 26036.126,E2 26036.126} C_VEL
LIN {X 0,Y 696.724,Z 1136.908,A -85,B 0,C 180,E1 26034.313,E2 26034.313} C_VEL
LIN {X 0,Y 696.401,Z 1151,A -85,B 0,C 180,E1 26032.008,E2 26032.008} C_VEL
LIN {X 0,Y 696.198,Z 1161.164,A -85,B 0,C 180,E1 26030.067,E2 26030.067} C_VEL
LIN {X 0,Y 696.07,Z 1169.059,A -85,B 0,C 180,E1 26028.335,E2 26028.335} C_VEL
LIN {X 0,Y 696.007,Z 1176.523,A -85,B 0,C 180,E1 26026.439,E2 26026.439} C_VEL
LIN {X 0,Y 695.947,Z 1183.578,A -85,B 0,C 180,E1 26024.222,E2 26024.222} C_VEL
LIN {X 0,Y 695.918,Z 1189.01,A -85,B 0,C 180,E1 26021.94,E2 26021.94} C_VEL
LIN {X 0,Y 695.908,Z 1192.462,A -85,B 0,C 180,E1 26019.844,E2 26019.844} C_VEL
LIN {X 0,Y 695.907,Z 1194.552,A -85,B 0,C 180,E1 26017.596,E2 26017.596} C_VEL
LIN {X 0,Y 695.895,Z 1194.866,A -85,B 0,C 180,E1 26015.441,E2 26015.441} C_VEL
LIN {X 0,Y 695.906,Z 1193.941,A -85,B 0,C 180,E1 26013.459,E2 26013.459} C_VEL
LIN {X 0,Y 695.911,Z 1191.269,A -85,B 0,C 180,E1 26011.235,E2 26011.235} C_VEL
LIN {X 0,Y 695.925,Z 1187.123,A -85,B 0,C 180,E1 26009.094,E2 26009.094} C_VEL
LIN {X 0,Y 695.961,Z 1181.411,A -85,B 0,C 180,E1 26006.953,E2 26006.953} C_VEL
LIN {X 0,Y 696.032,Z 1174.09,A -85,B 0,C 180,E1 26004.807,E2 26004.807} C_VEL
LIN {X 0,Y 696.151,Z 1163.897,A -85,B 0,C 180,E1 26002.407,E2 26002.407} C_VEL
LIN {X 0,Y 696.331,Z 1154.234,A -85,B 0,C 180,E1 26000.495,E2 26000.495} C_VEL
LIN {X 0,Y 696.539,Z 1144.145,A -85,B 0,C 180,E1 25998.742,E2 25998.742} C_VEL
LIN {X 0,Y 696.863,Z 1131.616,A -85,B 0,C 180,E1 25996.812,E2 25996.812} C_VEL
LIN {X 0,Y 697.338,Z 1115.27,A -85,B 0,C 180,E1 25994.617,E2 25994.617} C_VEL
LIN {X 0,Y 697.851,Z 1100.645,A -85,B 0,C 180,E1 25992.88,E2 25992.88} C_VEL
LIN {X 0,Y 698.511,Z 1082.606,A -85,B 0,C 180,E1 25990.951,E2 25990.951} C_VEL
LIN {X 0,Y 699.302,Z 1063.351,A -85,B 0,C 180,E1 25989.143,E2 25989.143} C_VEL
LIN {X 0,Y 700.025,Z 1045.993,A -85,B 0,C 180,E1 25987.67,E2 25987.67} C_VEL
LIN {X 0,Y 701.028,Z 1023.659,A -85,B 0,C 180,E1 25985.97,E2 25985.97} C_VEL
LIN {X 0,Y 701.928,Z 1003.447,A -85,B 0,C 180,E1 25984.61,E2 25984.61} C_VEL
LIN {X 0,Y 702.75,Z 985.214,A -85,B 0,C 180,E1 25983.504,E2 25983.504} C_VEL
LIN {X 0,Y 703.591,Z 965.985,A -85,B 0,C 180,E1 25982.451,E2 25982.451} C_VEL
LIN {X 0,Y 704.584,Z 943.047,A -85,B 0,C 180,E1 25981.337,E2 25981.337} C_VEL
LIN {X 0,Y 705.527,Z 917.193,A -85,B 0,C 180,E1 25980.263,E2 25980.263} C_VEL
LIN {X 0,Y 706.286,Z 895.658,A -85,B 0,C 180,E1 25979.501,E2 25979.501} C_VEL
LIN {X 0,Y 707.053,Z 873.084,A -85,B 0,C 180,E1 25978.82,E2 25978.82} C_VEL
LIN {X 0,Y 707.815,Z 845.649,A -85,B 0,C 180,E1 25978.158,E2 25978.158} C_VEL
LIN {X 0,Y 708.334,Z 818.882,A -85,B 0,C 180,E1 25977.683,E2 25977.683} C_VEL
LIN {X 0,Y 710.235,Z 598.546,A -85,B 0,C 180,E1 25974.945,E2 25974.945} C_VEL
LIN {X 0,Y 712.17,Z 377.545,A -85,B 0,C 180,E1 25972.125,E2 25972.125} C_VEL
LIN {X 0,Y 712.192,Z 357.963,A -85,B 0,C 180,E1 25971.858,E2 25971.858} C_VEL
LIN {X 0,Y 710.92,Z 353.964,A -85,B 0,C 180,E1 25971.704,E2 25971.704} C_VEL
LIN {X 0,Y 702.031,Z 340.419,A -85,B 0,C 180,E1 25970.774,E2 25970.774} C_VEL
LIN {X 0,Y 697.685,Z 330.946,A -85,B 0,C 180,E1 25969.68,E2 25969.68} C_VEL
LIN {X 0,Y 696.392,Z 327.488,A -85,B 0,C 180,E1 25969.264,E2 25969.264} C_VEL
LIN {X 0,Y 696.371,Z 327.489,A -85,B 0,C 180,E1 25966.319,E2 25966.319} C_VEL
LIN {X 0,Y 696.394,Z 327.484,A -85,B 0,C 180,E1 25963.405,E2 25963.405} C_VEL
LIN {X 0,Y 696.371,Z 327.489,A -85,B 0,C 180,E1 25960.448,E2 25960.448} C_VEL
LIN {X 0,Y 696.401,Z 327.478,A -85,B 0,C 180,E1 25957.501,E2 25957.501} C_VEL
LIN {X 0,Y 696.373,Z 327.488,A -85,B 0,C 180,E1 25954.453,E2 25954.453} C_VEL
LIN {X 0,Y 696.39,Z 327.481,A -85,B 0,C 180,E1 25951.51,E2 25951.51} C_VEL
LIN {X 0,Y 696.371,Z 327.482,A -85,B 0,C 180,E1 25948.377,E2 25948.377} C_VEL
LIN {X 0,Y 696.369,Z 327.47,A -85,B 0,C 180,E1 25945.516,E2 25945.516} C_VEL
LIN {X 0,Y 696.377,Z 327.481,A -85,B 0,C 180,E1 25942.365,E2 25942.365} C_VEL
LIN {X 0,Y 696.346,Z 327.471,A -85,B 0,C 180,E1 25939.619,E2 25939.619} C_VEL
LIN {X 0,Y 696.404,Z 327.485,A -85,B 0,C 180,E1 25936.688,E2 25936.688} C_VEL
LIN {X 0,Y 696.338,Z 327.467,A -85,B 0,C 180,E1 25933.79,E2 25933.79} C_VEL
LIN {X 0,Y 696.364,Z 327.481,A -85,B 0,C 180,E1 25931.093,E2 25931.093} C_VEL
LIN {X 0,Y 696.357,Z 327.488,A -85,B 0,C 180,E1 25928.006,E2 25928.006} C_VEL
LIN {X 0,Y 696.329,Z 327.482,A -85,B 0,C 180,E1 25925.356,E2 25925.356} C_VEL
LIN {X 0,Y 696.405,Z 327.485,A -85,B 0,C 180,E1 25922.469,E2 25922.469} C_VEL
LIN {X 0,Y 696.329,Z 327.488,A -85,B 0,C 180,E1 25919.589,E2 25919.589} C_VEL
LIN {X 0,Y 696.322,Z 327.486,A -85,B 0,C 180,E1 25917.119,E2 25917.119} C_VEL
LIN {X 0,Y 696.403,Z 327.482,A -85,B 0,C 180,E1 25914.232,E2 25914.232} C_VEL
LIN {X 0,Y 696.316,Z 327.485,A -85,B 0,C 180,E1 25911.411,E2 25911.411} C_VEL
LIN {X 0,Y 696.31,Z 327.488,A -85,B 0,C 180,E1 25908.99,E2 25908.99} C_VEL
LIN {X 0,Y 696.382,Z 327.468,A -85,B 0,C 180,E1 25906.211,E2 25906.211} C_VEL
LIN {X 0,Y 696.311,Z 327.491,A -85,B 0,C 180,E1 25903.293,E2 25903.293} C_VEL
LIN {X 0,Y 696.297,Z 327.478,A -85,B 0,C 180,E1 25900.888,E2 25900.888} C_VEL
LIN {X 0,Y 696.338,Z 327.486,A -85,B 0,C 180,E1 25898.255,E2 25898.255} C_VEL
LIN {X 0,Y 696.307,Z 327.473,A -85,B 0,C 180,E1 25895.209,E2 25895.209} C_VEL
LIN {X 0,Y 696.297,Z 327.491,A -85,B 0,C 180,E1 25892.733,E2 25892.733} C_VEL
LIN {X 0,Y 696.328,Z 327.489,A -85,B 0,C 180,E1 25890.209,E2 25890.209} C_VEL
LIN {X 0,Y 696.33,Z 327.491,A -85,B 0,C 180,E1 25887.126,E2 25887.126} C_VEL
LIN {X 0,Y 696.307,Z 327.492,A -85,B 0,C 180,E1 25884.64,E2 25884.64} C_VEL
LIN {X 0,Y 696.327,Z 327.493,A -85,B 0,C 180,E1 25882.163,E2 25882.163} C_VEL
LIN {X 0,Y 696.361,Z 327.49,A -85,B 0,C 180,E1 25879.098,E2 25879.098} C_VEL
LIN {X 0,Y 696.407,Z 327.533,A -85,B 0,C 180,E1 25877.398,E2 25877.398} C_VEL
LIN {X 0,Y 697.789,Z 331.161,A -85,B 0,C 180,E1 25876.993,E2 25876.993} C_VEL
LIN {X 0,Y 705.429,Z 347.653,A -85,B 0,C 180,E1 25875.099,E2 25875.099} C_VEL
LIN {X 0,Y 707.173,Z 351.342,A -85,B 0,C 180,E1 25874.724,E2 25874.724} C_VEL
LIN {X 0,Y 708.65,Z 354.322,A -85,B 0,C 180,E1 25874.565,E2 25874.565} C_VEL
LIN {X 0,Y 712.332,Z 368.798,A -85,B 0,C 180,E1 25874.074,E2 25874.074} C_VEL
LIN {X 0,Y 710.473,Z 579.67,A -85,B 0,C 180,E1 25871.374,E2 25871.374} C_VEL
LIN {X 0,Y 708.652,Z 803.091,A -85,B 0,C 180,E1 25868.605,E2 25868.605} C_VEL
LIN {X 0,Y 708.217,Z 836.687,A -85,B 0,C 180,E1 25868.151,E2 25868.151} C_VEL
LIN {X 0,Y 707.578,Z 863.534,A -85,B 0,C 180,E1 25867.623,E2 25867.623} C_VEL
LIN {X 0,Y 706.897,Z 888.651,A -85,B 0,C 180,E1 25866.981,E2 25866.981} C_VEL
LIN {X 0,Y 705.97,Z 916.879,A -85,B 0,C 180,E1 25866.072,E2 25866.072} C_VEL
LIN {X 0,Y 705.112,Z 939.367,A -85,B 0,C 180,E1 25865.205,E2 25865.205} C_VEL
LIN {X 0,Y 704.279,Z 959.698,A -85,B 0,C 180,E1 25864.307,E2 25864.307} C_VEL
LIN {X 0,Y 703.39,Z 980.311,A -85,B 0,C 180,E1 25863.278,E2 25863.278} C_VEL
LIN {X 0,Y 702.35,Z 1004.198,A -85,B 0,C 180,E1 25861.93,E2 25861.93} C_VEL
LIN {X 0,Y 701.361,Z 1026.243,A -85,B 0,C 180,E1 25860.499,E2 25860.499} C_VEL
LIN {X 0,Y 700.54,Z 1044.711,A -85,B 0,C 180,E1 25859.167,E2 25859.167} C_VEL
LIN {X 0,Y 699.648,Z 1065.139,A -85,B 0,C 180,E1 25857.537,E2 25857.537} C_VEL
LIN {X 0,Y 698.843,Z 1084.515,A -85,B 0,C 180,E1 25855.782,E2 25855.782} C_VEL
LIN {X 0,Y 698.207,Z 1100.539,A -85,B 0,C 180,E1 25854.178,E2 25854.178} C_VEL
LIN {X 0,Y 697.593,Z 1118.362,A -85,B 0,C 180,E1 25852.189,E2 25852.189} C_VEL
LIN {X 0,Y 697.09,Z 1133.808,A -85,B 0,C 180,E1 25850.224,E2 25850.224} C_VEL
LIN {X 0,Y 696.732,Z 1146.587,A -85,B 0,C 180,E1 25848.405,E2 25848.405} C_VEL
LIN {X 0,Y 696.412,Z 1159.875,A -85,B 0,C 180,E1 25846.259,E2 25846.259} C_VEL
LIN {X 0,Y 696.215,Z 1170.716,A -85,B 0,C 180,E1 25844.204,E2 25844.204} C_VEL
LIN {X 0,Y 696.087,Z 1178.791,A -85,B 0,C 180,E1 25842.443,E2 25842.443} C_VEL
LIN {X 0,Y 695.999,Z 1186.425,A -85,B 0,C 180,E1 25840.513,E2 25840.513} C_VEL
LIN {X 0,Y 695.948,Z 1193.594,A -85,B 0,C 180,E1 25838.261,E2 25838.261} C_VEL
LIN {X 0,Y 695.921,Z 1198.936,A -85,B 0,C 180,E1 25836.021,E2 25836.021} C_VEL
LIN {X 0,Y 695.909,Z 1202.483,A -85,B 0,C 180,E1 25833.872,E2 25833.872} C_VEL
LIN {X 0,Y 695.908,Z 1204.549,A -85,B 0,C 180,E1 25831.647,E2 25831.647} C_VEL
LIN {X 0,Y 695.89,Z 1204.872,A -85,B 0,C 180,E1 25829.506,E2 25829.506} C_VEL
LIN {X 0,Y 695.907,Z 1203.962,A -85,B 0,C 180,E1 25827.53,E2 25827.53} C_VEL
LIN {X 0,Y 695.909,Z 1201.428,A -85,B 0,C 180,E1 25825.385,E2 25825.385} C_VEL
LIN {X 0,Y 695.922,Z 1197.348,A -85,B 0,C 180,E1 25823.234,E2 25823.234} C_VEL
LIN {X 0,Y 695.957,Z 1191.391,A -85,B 0,C 180,E1 25820.991,E2 25820.991} C_VEL
LIN {X 0,Y 696.017,Z 1184.162,A -85,B 0,C 180,E1 25818.871,E2 25818.871} C_VEL
LIN {X 0,Y 696.165,Z 1173.94,A -85,B 0,C 180,E1 25816.461,E2 25816.461} C_VEL
LIN {X 0,Y 696.308,Z 1164.535,A -85,B 0,C 180,E1 25814.595,E2 25814.595} C_VEL
LIN {X 0,Y 696.535,Z 1154.749,A -85,B 0,C 180,E1 25812.886,E2 25812.886} C_VEL
LIN {X 0,Y 696.81,Z 1143.682,A -85,B 0,C 180,E1 25811.164,E2 25811.164} C_VEL
LIN {X 0,Y 697.257,Z 1128.618,A -85,B 0,C 180,E1 25809.08,E2 25809.08} C_VEL
LIN {X 0,Y 697.77,Z 1112.483,A -85,B 0,C 180,E1 25807.133,E2 25807.133} C_VEL
LIN {X 0,Y 698.355,Z 1097.131,A -85,B 0,C 180,E1 25805.468,E2 25805.468} C_VEL
LIN {X 0,Y 699.102,Z 1077.876,A -85,B 0,C 180,E1 25803.59,E2 25803.59} C_VEL
LIN {X 0,Y 699.907,Z 1059.058,A -85,B 0,C 180,E1 25801.966,E2 25801.966} C_VEL
LIN {X 0,Y 700.676,Z 1041.635,A -85,B 0,C 180,E1 25800.601,E2 25800.601} C_VEL
LIN {X 0,Y 701.655,Z 1019.539,A -85,B 0,C 180,E1 25799.041,E2 25799.041} C_VEL
LIN {X 0,Y 702.662,Z 997.046,A -85,B 0,C 180,E1 25797.654,E2 25797.654} C_VEL
LIN {X 0,Y 703.513,Z 977.652,A -85,B 0,C 180,E1 25796.583,E2 25796.583} C_VEL
LIN {X 0,Y 704.373,Z 957.726,A -85,B 0,C 180,E1 25795.6,E2 25795.6} C_VEL
LIN {X 0,Y 705.354,Z 933.847,A -85,B 0,C 180,E1 25794.566,E2 25794.566} C_VEL
LIN {X 0,Y 706.253,Z 907.061,A -85,B 0,C 180,E1 25793.591,E2 25793.591} C_VEL
LIN {X 0,Y 707.027,Z 883.672,A -85,B 0,C 180,E1 25792.881,E2 25792.881} C_VEL
LIN {X 0,Y 707.751,Z 857.844,A -85,B 0,C 180,E1 25792.251,E2 25792.251} C_VEL
LIN {X 0,Y 708.322,Z 830.084,A -85,B 0,C 180,E1 25791.745,E2 25791.745} C_VEL
LIN {X 0,Y 709.335,Z 716.686,A -85,B 0,C 180,E1 25790.334,E2 25790.334} C_VEL
LIN {X 0,Y 711.181,Z 498.02,A -85,B 0,C 180,E1 25787.592,E2 25787.592} C_VEL
LIN {X 0,Y 712.169,Z 367.486,A -85,B 0,C 180,E1 25785.895,E2 25785.895} C_VEL
LIN {X 0,Y 708.03,Z 352.73,A -85,B 0,C 180,E1 25785.364,E2 25785.364} C_VEL
LIN {X 0,Y 706.445,Z 350.088,A -85,B 0,C 180,E1 25785.163,E2 25785.163} C_VEL
LIN {X 0,Y 699.856,Z 335.529,A -85,B 0,C 180,E1 25783.523,E2 25783.523} C_VEL
LIN {X 0,Y 696.503,Z 328.118,A -85,B 0,C 180,E1 25782.656,E2 25782.656} C_VEL
LIN {X 0,Y 696.402,Z 327.489,A -85,B 0,C 180,E1 25782.562,E2 25782.562} C_VEL
LIN {X 0,Y 696.319,Z 327.493,A -85,B 0,C 180,E1 25779.677,E2 25779.677} C_VEL
LIN {X 0,Y 696.32,Z 327.489,A -85,B 0,C 180,E1 25777.196,E2 25777.196} C_VEL
LIN {X 0,Y 696.391,Z 327.488,A -85,B 0,C 180,E1 25774.253,E2 25774.253} C_VEL
LIN {X 0,Y 696.31,Z 327.484,A -85,B 0,C 180,E1 25771.466,E2 25771.466} C_VEL
LIN {X 0,Y 696.306,Z 327.488,A -85,B 0,C 180,E1 25769.131,E2 25769.131} C_VEL
LIN {X 0,Y 696.35,Z 327.478,A -85,B 0,C 180,E1 25766.524,E2 25766.524} C_VEL
LIN {X 0,Y 696.318,Z 327.489,A -85,B 0,C 180,E1 25763.528,E2 25763.528} C_VEL
LIN {X 0,Y 696.297,Z 327.481,A -85,B 0,C 180,E1 25761.127,E2 25761.127} C_VEL
LIN {X 0,Y 696.306,Z 327.491,A -85,B 0,C 180,E1 25758.677,E2 25758.677} C_VEL
LIN {X 0,Y 696.35,Z 327.484,A -85,B 0,C 180,E1 25755.661,E2 25755.661} C_VEL
LIN {X 0,Y 696.296,Z 327.488,A -85,B 0,C 180,E1 25753.03,E2 25753.03} C_VEL
LIN {X 0,Y 696.301,Z 327.478,A -85,B 0,C 180,E1 25750.592,E2 25750.592} C_VEL
LIN {X 0,Y 696.392,Z 327.482,A -85,B 0,C 180,E1 25747.674,E2 25747.674} C_VEL
LIN {X 0,Y 696.304,Z 327.483,A -85,B 0,C 180,E1 25744.86,E2 25744.86} C_VEL
LIN {X 0,Y 696.306,Z 327.49,A -85,B 0,C 180,E1 25742.469,E2 25742.469} C_VEL
LIN {X 0,Y 696.392,Z 327.472,A -85,B 0,C 180,E1 25739.671,E2 25739.671} C_VEL
LIN {X 0,Y 696.319,Z 327.487,A -85,B 0,C 180,E1 25736.79,E2 25736.79} C_VEL
LIN {X 0,Y 696.311,Z 327.474,A -85,B 0,C 180,E1 25734.314,E2 25734.314} C_VEL
LIN {X 0,Y 696.383,Z 327.49,A -85,B 0,C 180,E1 25731.578,E2 25731.578} C_VEL
LIN {X 0,Y 696.325,Z 327.481,A -85,B 0,C 180,E1 25728.57,E2 25728.57} C_VEL
LIN {X 0,Y 696.322,Z 327.488,A -85,B 0,C 180,E1 25726.093,E2 25726.093} C_VEL
LIN {X 0,Y 696.403,Z 327.476,A -85,B 0,C 180,E1 25723.226,E2 25723.226} C_VEL
LIN {X 0,Y 696.332,Z 327.478,A -85,B 0,C 180,E1 25720.366,E2 25720.366} C_VEL
LIN {X 0,Y 696.332,Z 327.487,A -85,B 0,C 180,E1 25717.812,E2 25717.812} C_VEL
LIN {X 0,Y 696.384,Z 327.475,A -85,B 0,C 180,E1 25715.258,E2 25715.258} C_VEL
LIN {X 0,Y 695.457,Z 327.595,A -85,B 0,C 180,E1 25714.624,E2 25714.624} C_VEL
LIN {X 0,Y 688.894,Z 328.42,A -85,B 0,C 180,E1 25712.804,E2 25712.804} C_VEL
LIN {X 0,Y 688.417,Z 328.473,A -85,B 0,C 180,E1 25712.387,E2 25712.387} C_VEL
LIN {X 0,Y 688.398,Z 328.475,A -85,B 0,C 180,E1 25709.734,E2 25709.734} C_VEL
LIN {X 0,Y 688.468,Z 328.476,A -85,B 0,C 180,E1 25706.802,E2 25706.802} C_VEL
LIN {X 0,Y 688.404,Z 328.481,A -85,B 0,C 180,E1 25703.858,E2 25703.858} C_VEL
LIN {X 0,Y 688.444,Z 328.612,A -85,B 0,C 180,E1 25703.228,E2 25703.228} C_VEL
LIN {X 0,Y 689.893,Z 332.136,A -85,B 0,C 180,E1 25702.816,E2 25702.816} C_VEL
LIN {X 0,Y 694.231,Z 341.402,A -85,B 0,C 180,E1 25701.746,E2 25701.746} C_VEL
LIN {X 0,Y 706.198,Z 359.533,A -85,B 0,C 180,E1 25700.503,E2 25700.503} C_VEL
LIN {X 0,Y 706.568,Z 362.182,A -85,B 0,C 180,E1 25700.436,E2 25700.436} C_VEL
LIN {X 0,Y 704.38,Z 578.779,A -85,B 0,C 180,E1 25697.645,E2 25697.645} C_VEL
LIN {X 0,Y 702.259,Z 807.184,A -85,B 0,C 180,E1 25694.795,E2 25694.795} C_VEL
LIN {X 0,Y 701.7,Z 834.483,A -85,B 0,C 180,E1 25694.373,E2 25694.373} C_VEL
LIN {X 0,Y 701.03,Z 859.446,A -85,B 0,C 180,E1 25693.843,E2 25693.843} C_VEL
LIN {X 0,Y 700.139,Z 886.392,A -85,B 0,C 180,E1 25693.106,E2 25693.106} C_VEL
LIN {X 0,Y 699.205,Z 910.43,A -85,B 0,C 180,E1 25692.29,E2 25692.29} C_VEL
LIN {X 0,Y 698.322,Z 931.129,A -85,B 0,C 180,E1 25691.474,E2 25691.474} C_VEL
LIN {X 0,Y 697.433,Z 950.474,A -85,B 0,C 180,E1 25690.607,E2 25690.607} C_VEL
LIN {X 0,Y 696.513,Z 969.402,A -85,B 0,C 180,E1 25689.655,E2 25689.655} C_VEL
LIN {X 0,Y 695.494,Z 989.948,A -85,B 0,C 180,E1 25688.499,E2 25688.499} C_VEL
LIN {X 0,Y 694.223,Z 1014.704,A -85,B 0,C 180,E1 25686.912,E2 25686.912} C_VEL
LIN {X 0,Y 693.287,Z 1033.293,A -85,B 0,C 180,E1 25685.567,E2 25685.567} C_VEL
LIN {X 0,Y 692.419,Z 1050.905,A -85,B 0,C 180,E1 25684.163,E2 25684.163} C_VEL
LIN {X 0,Y 691.423,Z 1071.367,A -85,B 0,C 180,E1 25682.348,E2 25682.348} C_VEL
LIN {X 0,Y 690.645,Z 1088.9,A -85,B 0,C 180,E1 25680.591,E2 25680.591} C_VEL
LIN {X 0,Y 689.986,Z 1104.573,A -85,B 0,C 180,E1 25678.852,E2 25678.852} C_VEL
LIN {X 0,Y 689.333,Z 1121.894,A -85,B 0,C 180,E1 25676.681,E2 25676.681} C_VEL
LIN {X 0,Y 688.906,Z 1135.112,A -85,B 0,C 180,E1 25674.8,E2 25674.8} C_VEL
LIN {X 0,Y 688.57,Z 1146.976,A -85,B 0,C 180,E1 25672.902,E2 25672.902} C_VEL
LIN {X 0,Y 688.297,Z 1159.499,A -85,B 0,C 180,E1 25670.582,E2 25670.582} C_VEL
LIN {X 0,Y 688.128,Z 1168.382,A -85,B 0,C 180,E1 25668.642,E2 25668.642} C_VEL
LIN {X 0,Y 688.021,Z 1176.265,A -85,B 0,C 180,E1 25666.636,E2 25666.636} C_VEL
LIN {X 0,Y 687.959,Z 1183.37,A -85,B 0,C 180,E1 25664.39,E2 25664.39} C_VEL
LIN {X 0,Y 687.923,Z 1188.69,A -85,B 0,C 180,E1 25662.166,E2 25662.166} C_VEL
LIN {X 0,Y 687.912,Z 1192.255,A -85,B 0,C 180,E1 25660.044,E2 25660.044} C_VEL
LIN {X 0,Y 687.906,Z 1194.45,A -85,B 0,C 180,E1 25657.768,E2 25657.768} C_VEL
LIN {X 0,Y 687.892,Z 1194.885,A -85,B 0,C 180,E1 25655.505,E2 25655.505} C_VEL
LIN {X 0,Y 687.906,Z 1193.995,A -85,B 0,C 180,E1 25653.5,E2 25653.5} C_VEL
LIN {X 0,Y 687.91,Z 1191.497,A -85,B 0,C 180,E1 25651.332,E2 25651.332} C_VEL
LIN {X 0,Y 687.928,Z 1187.285,A -85,B 0,C 180,E1 25649.084,E2 25649.084} C_VEL
LIN {X 0,Y 687.971,Z 1181.368,A -85,B 0,C 180,E1 25646.834,E2 25646.834} C_VEL
LIN {X 0,Y 688.053,Z 1174.041,A -85,B 0,C 180,E1 25644.663,E2 25644.663} C_VEL
LIN {X 0,Y 688.184,Z 1163.837,A -85,B 0,C 180,E1 25642.234,E2 25642.234} C_VEL
LIN {X 0,Y 688.407,Z 1154.169,A -85,B 0,C 180,E1 25640.3,E2 25640.3} C_VEL
LIN {X 0,Y 688.645,Z 1144.074,A -85,B 0,C 180,E1 25638.526,E2 25638.526} C_VEL
LIN {X 0,Y 689.035,Z 1130.974,A -85,B 0,C 180,E1 25636.489,E2 25636.489} C_VEL
LIN {X 0,Y 689.575,Z 1114.957,A -85,B 0,C 180,E1 25634.325,E2 25634.325} C_VEL
LIN {X 0,Y 690.175,Z 1100.132,A -85,B 0,C 180,E1 25632.549,E2 25632.549} C_VEL
LIN {X 0,Y 690.966,Z 1081.601,A -85,B 0,C 180,E1 25630.559,E2 25630.559} C_VEL
LIN {X 0,Y 691.806,Z 1063.228,A -85,B 0,C 180,E1 25628.818,E2 25628.818} C_VEL
LIN {X 0,Y 692.637,Z 1045.858,A -85,B 0,C 180,E1 25627.329,E2 25627.329} C_VEL
LIN {X 0,Y 693.793,Z 1023.617,A -85,B 0,C 180,E1 25625.622,E2 25625.622} C_VEL
LIN {X 0,Y 694.79,Z 1003.823,A -85,B 0,C 180,E1 25624.276,E2 25624.276} C_VEL
LIN {X 0,Y 695.741,Z 985.102,A -85,B 0,C 180,E1 25623.129,E2 25623.129} C_VEL
LIN {X 0,Y 696.662,Z 966.512,A -85,B 0,C 180,E1 25622.102,E2 25622.102} C_VEL
LIN {X 0,Y 697.672,Z 945.616,A -85,B 0,C 180,E1 25621.073,E2 25621.073} C_VEL
LIN {X 0,Y 698.812,Z 919.237,A -85,B 0,C 180,E1 25619.948,E2 25619.948} C_VEL
LIN {X 0,Y 699.734,Z 895.925,A -85,B 0,C 180,E1 25619.113,E2 25619.113} C_VEL
LIN {X 0,Y 700.584,Z 873.499,A -85,B 0,C 180,E1 25618.432,E2 25618.432} C_VEL
LIN {X 0,Y 701.426,Z 846.493,A -85,B 0,C 180,E1 25617.772,E2 25617.772} C_VEL
LIN {X 0,Y 702.028,Z 819.578,A -85,B 0,C 180,E1 25617.287,E2 25617.287} C_VEL
LIN {X 0,Y 703.158,Z 707.993,A -85,B 0,C 180,E1 25615.888,E2 25615.888} C_VEL
LIN {X 0,Y 705.113,Z 500.579,A -85,B 0,C 180,E1 25613.266,E2 25613.266} C_VEL
LIN {X 0,Y 706.437,Z 360.31,A -85,B 0,C 180,E1 25611.437,E2 25611.437} C_VEL
LIN {X 0,Y 705.407,Z 357.986,A -85,B 0,C 180,E1 25611.322,E2 25611.322} C_VEL
LIN {X 0,Y 693.896,Z 340.702,A -85,B 0,C 180,E1 25610.116,E2 25610.116} C_VEL
LIN {X 0,Y 689.697,Z 331.85,A -85,B 0,C 180,E1 25609.054,E2 25609.054} C_VEL
LIN {X 0,Y 688.44,Z 328.475,A -85,B 0,C 180,E1 25608.636,E2 25608.636} C_VEL
LIN {X 0,Y 688.463,Z 328.474,A -85,B 0,C 180,E1 25605.687,E2 25605.687} C_VEL
LIN {X 0,Y 688.44,Z 328.478,A -85,B 0,C 180,E1 25602.596,E2 25602.596} C_VEL
LIN {X 0,Y 688.462,Z 328.471,A -85,B 0,C 180,E1 25599.612,E2 25599.612} C_VEL
LIN {X 0,Y 688.44,Z 328.477,A -85,B 0,C 180,E1 25596.547,E2 25596.547} C_VEL
LIN {X 0,Y 688.448,Z 328.47,A -85,B 0,C 180,E1 25593.598,E2 25593.598} C_VEL
LIN {X 0,Y 688.438,Z 328.475,A -85,B 0,C 180,E1 25590.457,E2 25590.457} C_VEL
LIN {X 0,Y 688.429,Z 328.464,A -85,B 0,C 180,E1 25587.602,E2 25587.602} C_VEL
LIN {X 0,Y 688.445,Z 328.474,A -85,B 0,C 180,E1 25584.452,E2 25584.452} C_VEL
LIN {X 0,Y 688.411,Z 328.465,A -85,B 0,C 180,E1 25581.633,E2 25581.633} C_VEL
LIN {X 0,Y 688.464,Z 328.462,A -85,B 0,C 180,E1 25578.634,E2 25578.634} C_VEL
LIN {X 0,Y 688.403,Z 328.469,A -85,B 0,C 180,E1 25575.76,E2 25575.76} C_VEL
LIN {X 0,Y 688.451,Z 328.449,A -85,B 0,C 180,E1 25572.925,E2 25572.925} C_VEL
LIN {X 0,Y 688.405,Z 328.475,A -85,B 0,C 180,E1 25569.869,E2 25569.869} C_VEL
LIN {X 0,Y 688.401,Z 328.474,A -85,B 0,C 180,E1 25567.237,E2 25567.237} C_VEL
LIN {X 0,Y 688.455,Z 328.474,A -85,B 0,C 180,E1 25564.248,E2 25564.248} C_VEL
LIN {X 0,Y 688.386,Z 328.472,A -85,B 0,C 180,E1 25561.498,E2 25561.498} C_VEL
LIN {X 0,Y 688.401,Z 328.475,A -85,B 0,C 180,E1 25558.918,E2 25558.918} C_VEL
LIN {X 0,Y 688.404,Z 328.476,A -85,B 0,C 180,E1 25555.752,E2 25555.752} C_VEL
LIN {X 0,Y 688.376,Z 328.477,A -85,B 0,C 180,E1 25553.159,E2 25553.159} C_VEL
LIN {X 0,Y 688.409,Z 328.472,A -85,B 0,C 180,E1 25550.553,E2 25550.553} C_VEL
LIN {X 0,Y 688.385,Z 328.464,A -85,B 0,C 180,E1 25547.501,E2 25547.501} C_VEL
LIN {X 0,Y 688.365,Z 328.472,A -85,B 0,C 180,E1 25545.003,E2 25545.003} C_VEL
LIN {X 0,Y 688.396,Z 328.479,A -85,B 0,C 180,E1 25542.415,E2 25542.415} C_VEL
LIN {X 0,Y 688.374,Z 328.475,A -85,B 0,C 180,E1 25539.297,E2 25539.297} C_VEL
LIN {X 0,Y 688.355,Z 328.48,A -85,B 0,C 180,E1 25536.849,E2 25536.849} C_VEL
LIN {X 0,Y 688.385,Z 328.459,A -85,B 0,C 180,E1 25534.259,E2 25534.259} C_VEL
LIN {X 0,Y 688.377,Z 328.478,A -85,B 0,C 180,E1 25531.148,E2 25531.148} C_VEL
LIN {X 0,Y 688.363,Z 328.476,A -85,B 0,C 180,E1 25528.764,E2 25528.764} C_VEL
LIN {X 0,Y 688.378,Z 328.482,A -85,B 0,C 180,E1 25526.298,E2 25526.298} C_VEL
LIN {X 0,Y 688.43,Z 328.48,A -85,B 0,C 180,E1 25523.295,E2 25523.295} C_VEL
LIN {X 0,Y 688.376,Z 328.485,A -85,B 0,C 180,E1 25520.598,E2 25520.598} C_VEL
LIN {X 0,Y 688.393,Z 328.478,A -85,B 0,C 180,E1 25518.059,E2 25518.059} C_VEL
LIN {X 0,Y 689.872,Z 332.132,A -85,B 0,C 180,E1 25517.626,E2 25517.626} C_VEL
LIN {X 0,Y 698.081,Z 349.885,A -85,B 0,C 180,E1 25515.539,E2 25515.539} C_VEL
LIN {X 0,Y 699.256,Z 351.999,A -85,B 0,C 180,E1 25515.361,E2 25515.361} C_VEL
LIN {X 0,Y 703.374,Z 358.356,A -85,B 0,C 180,E1 25514.932,E2 25514.932} C_VEL
LIN {X 0,Y 706.55,Z 371.037,A -85,B 0,C 180,E1 25514.499,E2 25514.499} C_VEL
LIN {X 0,Y 704.436,Z 582.331,A -85,B 0,C 180,E1 25511.772,E2 25511.772} C_VEL
LIN {X 0,Y 702.374,Z 805.259,A -85,B 0,C 180,E1 25508.988,E2 25508.988} C_VEL
LIN {X 0,Y 701.874,Z 837.902,A -85,B 0,C 180,E1 25508.535,E2 25508.535} C_VEL
LIN {X 0,Y 701.176,Z 864.088,A -85,B 0,C 180,E1 25508.013,E2 25508.013} C_VEL
LIN {X 0,Y 700.402,Z 889.168,A -85,B 0,C 180,E1 25507.366,E2 25507.366} C_VEL
LIN {X 0,Y 699.348,Z 917.454,A -85,B 0,C 180,E1 25506.445,E2 25506.445} C_VEL
LIN {X 0,Y 698.407,Z 939.443,A -85,B 0,C 180,E1 25505.591,E2 25505.591} C_VEL
LIN {X 0,Y 697.474,Z 959.701,A -85,B 0,C 180,E1 25504.69,E2 25504.69} C_VEL
LIN {X 0,Y 696.516,Z 979.424,A -85,B 0,C 180,E1 25503.7,E2 25503.7} C_VEL
LIN {X 0,Y 695.398,Z 1001.889,A -85,B 0,C 180,E1 25502.432,E2 25502.432} C_VEL
LIN {X 0,Y 694.217,Z 1024.91,A -85,B 0,C 180,E1 25500.943,E2 25500.943} C_VEL
LIN {X 0,Y 693.267,Z 1043.782,A -85,B 0,C 180,E1 25499.576,E2 25499.576} C_VEL
LIN {X 0,Y 692.352,Z 1062.371,A -85,B 0,C 180,E1 25498.087,E2 25498.087} C_VEL
LIN {X 0,Y 691.306,Z 1083.584,A -85,B 0,C 180,E1 25496.177,E2 25496.177} C_VEL
LIN {X 0,Y 690.611,Z 1099.687,A -85,B 0,C 180,E1 25494.552,E2 25494.552} C_VEL
LIN {X 0,Y 689.909,Z 1116.488,A -85,B 0,C 180,E1 25492.676,E2 25492.676} C_VEL
LIN {X 0,Y 689.313,Z 1132.52,A -85,B 0,C 180,E1 25490.639,E2 25490.639} C_VEL
LIN {X 0,Y 688.907,Z 1145.025,A -85,B 0,C 180,E1 25488.857,E2 25488.857} C_VEL
LIN {X 0,Y 688.592,Z 1156.312,A -85,B 0,C 180,E1 25487.057,E2 25487.057} C_VEL
LIN {X 0,Y 688.307,Z 1168.604,A -85,B 0,C 180,E1 25484.813,E2 25484.813} C_VEL
LIN {X 0,Y 688.132,Z 1178.077,A -85,B 0,C 180,E1 25482.76,E2 25482.76} C_VEL
LIN {X 0,Y 688.006,Z 1186.016,A -85,B 0,C 180,E1 25480.751,E2 25480.751} C_VEL
LIN {X 0,Y 687.958,Z 1193.109,A -85,B 0,C 180,E1 25478.526,E2 25478.526} C_VEL
LIN {X 0,Y 687.927,Z 1198.593,A -85,B 0,C 180,E1 25476.259,E2 25476.259} C_VEL
LIN {X 0,Y 687.915,Z 1202.263,A -85,B 0,C 180,E1 25474.084,E2 25474.084} C_VEL
LIN {X 0,Y 687.907,Z 1204.437,A -85,B 0,C 180,E1 25471.833,E2 25471.833} C_VEL
LIN {X 0,Y 687.891,Z 1204.894,A -85,B 0,C 180,E1 25469.584,E2 25469.584} C_VEL
LIN {X 0,Y 687.907,Z 1203.959,A -85,B 0,C 180,E1 25467.501,E2 25467.501} C_VEL
LIN {X 0,Y 687.911,Z 1201.428,A -85,B 0,C 180,E1 25465.332,E2 25465.332} C_VEL
LIN {X 0,Y 687.928,Z 1197.152,A -85,B 0,C 180,E1 25463.071,E2 25463.071} C_VEL
LIN {X 0,Y 687.967,Z 1191.388,A -85,B 0,C 180,E1 25460.885,E2 25460.885} C_VEL
LIN {X 0,Y 688.039,Z 1184.278,A -85,B 0,C 180,E1 25458.771,E2 25458.771} C_VEL
LIN {X 0,Y 688.2,Z 1173.939,A -85,B 0,C 180,E1 25456.301,E2 25456.301} C_VEL
LIN {X 0,Y 688.395,Z 1164.292,A -85,B 0,C 180,E1 25454.368,E2 25454.368} C_VEL
LIN {X 0,Y 688.644,Z 1154.228,A -85,B 0,C 180,E1 25452.597,E2 25452.597} C_VEL
LIN {X 0,Y 688.983,Z 1142.519,A -85,B 0,C 180,E1 25450.766,E2 25450.766} C_VEL
LIN {X 0,Y 689.531,Z 1126.514,A -85,B 0,C 180,E1 25448.567,E2 25448.567} C_VEL
LIN {X 0,Y 690.12,Z 1111.234,A -85,B 0,C 180,E1 25446.72,E2 25446.72} C_VEL
LIN {X 0,Y 690.811,Z 1094.572,A -85,B 0,C 180,E1 25444.908,E2 25444.908} C_VEL
LIN {X 0,Y 691.751,Z 1074.835,A -85,B 0,C 180,E1 25443.009,E2 25443.009} C_VEL
LIN {X 0,Y 692.544,Z 1057.951,A -85,B 0,C 180,E1 25441.547,E2 25441.547} C_VEL
LIN {X 0,Y 693.497,Z 1038.972,A -85,B 0,C 180,E1 25440.058,E2 25440.058} C_VEL
LIN {X 0,Y 694.719,Z 1015.175,A -85,B 0,C 180,E1 25438.407,E2 25438.407} C_VEL
LIN {X 0,Y 695.721,Z 995.443,A -85,B 0,C 180,E1 25437.193,E2 25437.193} C_VEL
LIN {X 0,Y 696.698,Z 975.872,A -85,B 0,C 180,E1 25436.113,E2 25436.113} C_VEL
LIN {X 0,Y 697.765,Z 953.703,A -85,B 0,C 180,E1 25435.028,E2 25435.028} C_VEL
LIN {X 0,Y 698.897,Z 927.095,A -85,B 0,C 180,E1 25433.911,E2 25433.911} C_VEL
LIN {X 0,Y 699.79,Z 904.867,A -85,B 0,C 180,E1 25433.123,E2 25433.123} C_VEL
LIN {X 0,Y 700.638,Z 881.835,A -85,B 0,C 180,E1 25432.431,E2 25432.431} C_VEL
LIN {X 0,Y 701.466,Z 854.971,A -85,B 0,C 180,E1 25431.785,E2 25431.785} C_VEL
LIN {X 0,Y 702.071,Z 827.525,A -85,B 0,C 180,E1 25431.303,E2 25431.303} C_VEL
LIN {X 0,Y 704.226,Z 604.152,A -85,B 0,C 180,E1 25428.505,E2 25428.505} C_VEL
LIN {X 0,Y 706.242,Z 400.121,A -85,B 0,C 180,E1 25425.882,E2 25425.882} C_VEL
LIN {X 0,Y 706.388,Z 369.725,A -85,B 0,C 180,E1 25425.47,E2 25425.47} C_VEL
LIN {X 0,Y 702.932,Z 357.34,A -85,B 0,C 180,E1 25425.017,E2 25425.017} C_VEL
LIN {X 0,Y 698.283,Z 350.368,A -85,B 0,C 180,E1 25424.514,E2 25424.514} C_VEL
LIN {X 0,Y 691.523,Z 335.795,A -85,B 0,C 180,E1 25422.811,E2 25422.811} C_VEL
LIN {X 0,Y 689.872,Z 332.132,A -85,B 0,C 180,E1 25422.374,E2 25422.374} C_VEL
LIN {X 0,Y 688.412,Z 328.583,A -85,B 0,C 180,E1 25421.958,E2 25421.958} C_VEL
LIN {X 0,Y 688.377,Z 328.482,A -85,B 0,C 180,E1 25419.401,E2 25419.401} C_VEL
LIN {X 0,Y 688.439,Z 328.476,A -85,B 0,C 180,E1 25416.651,E2 25416.651} C_VEL
LIN {X 0,Y 688.382,Z 328.479,A -85,B 0,C 180,E1 25413.667,E2 25413.667} C_VEL
LIN {X 0,Y 688.37,Z 328.472,A -85,B 0,C 180,E1 25411.182,E2 25411.182} C_VEL
LIN {X 0,Y 688.422,Z 328.477,A -85,B 0,C 180,E1 25408.514,E2 25408.514} C_VEL
LIN {X 0,Y 688.381,Z 328.476,A -85,B 0,C 180,E1 25405.557,E2 25405.557} C_VEL
LIN {X 0,Y 688.36,Z 328.478,A -85,B 0,C 180,E1 25403.091,E2 25403.091} C_VEL
LIN {X 0,Y 688.373,Z 328.469,A -85,B 0,C 180,E1 25400.669,E2 25400.669} C_VEL
LIN {X 0,Y 688.394,Z 328.467,A -85,B 0,C 180,E1 25397.585,E2 25397.585} C_VEL
LIN {X 0,Y 688.353,Z 328.478,A -85,B 0,C 180,E1 25394.985,E2 25394.985} C_VEL
LIN {X 0,Y 688.365,Z 328.477,A -85,B 0,C 180,E1 25392.553,E2 25392.553} C_VEL
LIN {X 0,Y 688.429,Z 328.476,A -85,B 0,C 180,E1 25389.615,E2 25389.615} C_VEL
LIN {X 0,Y 688.366,Z 328.471,A -85,B 0,C 180,E1 25386.925,E2 25386.925} C_VEL
LIN {X 0,Y 688.366,Z 328.472,A -85,B 0,C 180,E1 25384.499,E2 25384.499} C_VEL
LIN {X 0,Y 688.459,Z 328.463,A -85,B 0,C 180,E1 25381.581,E2 25381.581} C_VEL
LIN {X 0,Y 688.374,Z 328.475,A -85,B 0,C 180,E1 25378.752,E2 25378.752} C_VEL
LIN {X 0,Y 688.375,Z 328.477,A -85,B 0,C 180,E1 25376.252,E2 25376.252} C_VEL
LIN {X 0,Y 688.462,Z 328.469,A -85,B 0,C 180,E1 25373.328,E2 25373.328} C_VEL
LIN {X 0,Y 688.377,Z 328.47,A -85,B 0,C 180,E1 25370.469,E2 25370.469} C_VEL
LIN {X 0,Y 688.393,Z 328.471,A -85,B 0,C 180,E1 25367.927,E2 25367.927} C_VEL
LIN {X 0,Y 688.424,Z 328.456,A -85,B 0,C 180,E1 25364.844,E2 25364.844} C_VEL
LIN {X 0,Y 688.386,Z 328.476,A -85,B 0,C 180,E1 25362.153,E2 25362.153} C_VEL
LIN {X 0,Y 688.433,Z 328.461,A -85,B 0,C 180,E1 25359.422,E2 25359.422} C_VEL
LIN {X 0,Y 688.404,Z 328.47,A -85,B 0,C 180,E1 25356.366,E2 25356.366} C_VEL
LIN {X 0,Y 688.395,Z 328.475,A -85,B 0,C 180,E1 25353.796,E2 25353.796} C_VEL
LIN {X 0,Y 688.417,Z 328.473,A -85,B 0,C 180,E1 25352.387,E2 25352.387} C_VEL
LIN {X 0,Y 687.378,Z 328.603,A -85,B 0,C 180,E1 25351.746,E2 25351.746} C_VEL
LIN {X 0,Y 680.965,Z 329.401,A -85,B 0,C 180,E1 25349.949,E2 25349.949} C_VEL
LIN {X 0,Y 680.471,Z 329.465,A -85,B 0,C 180,E1 25349.482,E2 25349.482} C_VEL
LIN {X 0,Y 680.497,Z 329.465,A -85,B 0,C 180,E1 25346.362,E2 25346.362} C_VEL
LIN {X 0,Y 680.48,Z 329.568,A -85,B 0,C 180,E1 25343.881,E2 25343.881} C_VEL
LIN {X 0,Y 681.872,Z 333.093,A -85,B 0,C 180,E1 25343.462,E2 25343.462} C_VEL
LIN {X 0,Y 685.875,Z 341.383,A -85,B 0,C 180,E1 25342.469,E2 25342.469} C_VEL
LIN {X 0,Y 698.969,Z 360.812,A -85,B 0,C 180,E1 25341.071,E2 25341.071} C_VEL
LIN {X 0,Y 700.83,Z 363.986,A -85,B 0,C 180,E1 25340.873,E2 25340.873} C_VEL
LIN {X 0,Y 698.376,Z 580.896,A -85,B 0,C 180,E1 25338.056,E2 25338.056} C_VEL
LIN {X 0,Y 695.981,Z 809.656,A -85,B 0,C 180,E1 25335.177,E2 25335.177} C_VEL
LIN {X 0,Y 695.371,Z 835.626,A -85,B 0,C 180,E1 25334.763,E2 25334.763} C_VEL
LIN {X 0,Y 694.62,Z 860.817,A -85,B 0,C 180,E1 25334.219,E2 25334.219} C_VEL
LIN {X 0,Y 693.609,Z 887.588,A -85,B 0,C 180,E1 25333.473,E2 25333.473} C_VEL
LIN {X 0,Y 692.612,Z 910.843,A -85,B 0,C 180,E1 25332.676,E2 25332.676} C_VEL
LIN {X 0,Y 691.685,Z 930.401,A -85,B 0,C 180,E1 25331.901,E2 25331.901} C_VEL
LIN {X 0,Y 690.706,Z 949.521,A -85,B 0,C 180,E1 25331.042,E2 25331.042} C_VEL
LIN {X 0,Y 689.66,Z 968.813,A -85,B 0,C 180,E1 25330.069,E2 25330.069} C_VEL
LIN {X 0,Y 688.567,Z 988.47,A -85,B 0,C 180,E1 25328.958,E2 25328.958} C_VEL
LIN {X 0,Y 687.206,Z 1012.061,A -85,B 0,C 180,E1 25327.458,E2 25327.458} C_VEL
LIN {X 0,Y 686.032,Z 1032.575,A -85,B 0,C 180,E1 25325.97,E2 25325.97} C_VEL
LIN {X 0,Y 685.056,Z 1050.324,A -85,B 0,C 180,E1 25324.543,E2 25324.543} C_VEL
LIN {X 0,Y 683.97,Z 1070.514,A -85,B 0,C 180,E1 25322.744,E2 25322.744} C_VEL
LIN {X 0,Y 683.031,Z 1088.586,A -85,B 0,C 180,E1 25320.918,E2 25320.918} C_VEL
LIN {X 0,Y 682.279,Z 1104.471,A -85,B 0,C 180,E1 25319.138,E2 25319.138} C_VEL
LIN {X 0,Y 681.545,Z 1121.694,A -85,B 0,C 180,E1 25316.957,E2 25316.957} C_VEL
LIN {X 0,Y 681.06,Z 1134.869,A -85,B 0,C 180,E1 25315.063,E2 25315.063} C_VEL
LIN {X 0,Y 680.686,Z 1146.517,A -85,B 0,C 180,E1 25313.183,E2 25313.183} C_VEL
LIN {X 0,Y 680.36,Z 1159.201,A -85,B 0,C 180,E1 25310.82,E2 25310.82} C_VEL
LIN {X 0,Y 680.163,Z 1168.439,A -85,B 0,C 180,E1 25308.78,E2 25308.78} C_VEL
LIN {X 0,Y 680.034,Z 1176.311,A -85,B 0,C 180,E1 25306.749,E2 25306.749} C_VEL
LIN {X 0,Y 679.968,Z 1183.41,A -85,B 0,C 180,E1 25304.476,E2 25304.476} C_VEL
LIN {X 0,Y 679.923,Z 1188.894,A -85,B 0,C 180,E1 25302.139,E2 25302.139} C_VEL
LIN {X 0,Y 679.911,Z 1192.387,A -85,B 0,C 180,E1 25299.993,E2 25299.993} C_VEL
LIN {X 0,Y 679.906,Z 1194.516,A -85,B 0,C 180,E1 25297.69,E2 25297.69} C_VEL
LIN {X 0,Y 679.893,Z 1194.881,A -85,B 0,C 180,E1 25295.485,E2 25295.485} C_VEL
LIN {X 0,Y 679.906,Z 1193.98,A -85,B 0,C 180,E1 25293.456,E2 25293.456} C_VEL
LIN {X 0,Y 679.912,Z 1191.477,A -85,B 0,C 180,E1 25291.264,E2 25291.264} C_VEL
LIN {X 0,Y 679.935,Z 1187.253,A -85,B 0,C 180,E1 25288.989,E2 25288.989} C_VEL
LIN {X 0,Y 679.982,Z 1181.325,A -85,B 0,C 180,E1 25286.712,E2 25286.712} C_VEL
LIN {X 0,Y 680.076,Z 1173.883,A -85,B 0,C 180,E1 25284.486,E2 25284.486} C_VEL
LIN {X 0,Y 680.227,Z 1163.776,A -85,B 0,C 180,E1 25282.058,E2 25282.058} C_VEL
LIN {X 0,Y 680.478,Z 1154.105,A -85,B 0,C 180,E1 25280.1,E2 25280.1} C_VEL
LIN {X 0,Y 680.764,Z 1144.004,A -85,B 0,C 180,E1 25278.306,E2 25278.306} C_VEL
LIN {X 0,Y 681.225,Z 1130.333,A -85,B 0,C 180,E1 25276.158,E2 25276.158} C_VEL
LIN {X 0,Y 681.842,Z 1114.403,A -85,B 0,C 180,E1 25273.997,E2 25273.997} C_VEL
LIN {X 0,Y 682.485,Z 1099.823,A -85,B 0,C 180,E1 25272.233,E2 25272.233} C_VEL
LIN {X 0,Y 683.454,Z 1080.595,A -85,B 0,C 180,E1 25270.159,E2 25270.159} C_VEL
LIN {X 0,Y 684.331,Z 1063.105,A -85,B 0,C 180,E1 25268.485,E2 25268.485} C_VEL
LIN {X 0,Y 685.278,Z 1045.723,A -85,B 0,C 180,E1 25266.981,E2 25266.981} C_VEL
LIN {X 0,Y 686.627,Z 1022.696,A -85,B 0,C 180,E1 25265.204,E2 25265.204} C_VEL
LIN {X 0,Y 687.733,Z 1003.08,A -85,B 0,C 180,E1 25263.862,E2 25263.862} C_VEL
LIN {X 0,Y 688.804,Z 984.133,A -85,B 0,C 180,E1 25262.696,E2 25262.696} C_VEL
LIN {X 0,Y 689.981,Z 962.875,A -85,B 0,C 180,E1 25261.525,E2 25261.525} C_VEL
LIN {X 0,Y 691.379,Z 936.311,A -85,B 0,C 180,E1 25260.261,E2 25260.261} C_VEL
LIN {X 0,Y 692.394,Z 915.126,A -85,B 0,C 180,E1 25259.394,E2 25259.394} C_VEL
LIN {X 0,Y 693.274,Z 894.805,A -85,B 0,C 180,E1 25258.672,E2 25258.672} C_VEL
LIN {X 0,Y 694.221,Z 872.15,A -85,B 0,C 180,E1 25257.987,E2 25257.987} C_VEL
LIN {X 0,Y 695.146,Z 844.744,A -85,B 0,C 180,E1 25257.324,E2 25257.324} C_VEL
LIN {X 0,Y 695.798,Z 818.104,A -85,B 0,C 180,E1 25256.853,E2 25256.853} C_VEL
LIN {X 0,Y 698.169,Z 600.288,A -85,B 0,C 180,E1 25254.101,E2 25254.101} C_VEL
LIN {X 0,Y 700.635,Z 379.143,A -85,B 0,C 180,E1 25251.236,E2 25251.236} C_VEL
LIN {X 0,Y 700.71,Z 363.362,A -85,B 0,C 180,E1 25251.018,E2 25251.018} C_VEL
LIN {X 0,Y 688.105,Z 344.783,A -85,B 0,C 180,E1 25249.687,E2 25249.687} C_VEL
LIN {X 0,Y 685.298,Z 340.451,A -85,B 0,C 180,E1 25249.351,E2 25249.351} C_VEL
LIN {X 0,Y 681.745,Z 332.861,A -85,B 0,C 180,E1 25248.418,E2 25248.418} C_VEL
LIN {X 0,Y 680.513,Z 329.457,A -85,B 0,C 180,E1 25247.995,E2 25247.995} C_VEL
LIN {X 0,Y 680.515,Z 329.466,A -85,B 0,C 180,E1 25244.792,E2 25244.792} C_VEL
LIN {X 0,Y 680.522,Z 329.458,A -85,B 0,C 180,E1 25241.721,E2 25241.721} C_VEL
LIN {X 0,Y 680.503,Z 329.465,A -85,B 0,C 180,E1 25238.585,E2 25238.585} C_VEL
LIN {X 0,Y 680.517,Z 329.457,A -85,B 0,C 180,E1 25235.581,E2 25235.581} C_VEL
LIN {X 0,Y 680.496,Z 329.467,A -85,B 0,C 180,E1 25232.433,E2 25232.433} C_VEL
LIN {X 0,Y 680.505,Z 329.459,A -85,B 0,C 180,E1 25229.487,E2 25229.487} C_VEL
LIN {X 0,Y 680.489,Z 329.444,A -85,B 0,C 180,E1 25226.323,E2 25226.323} C_VEL
LIN {X 0,Y 680.49,Z 329.461,A -85,B 0,C 180,E1 25223.466,E2 25223.466} C_VEL
LIN {X 0,Y 680.49,Z 329.442,A -85,B 0,C 180,E1 25220.29,E2 25220.29} C_VEL
LIN {X 0,Y 680.473,Z 329.462,A -85,B 0,C 180,E1 25217.516,E2 25217.516} C_VEL
LIN {X 0,Y 680.522,Z 329.439,A -85,B 0,C 180,E1 25214.465,E2 25214.465} C_VEL
LIN {X 0,Y 680.459,Z 329.461,A -85,B 0,C 180,E1 25211.614,E2 25211.614} C_VEL
LIN {X 0,Y 680.524,Z 329.459,A -85,B 0,C 180,E1 25208.704,E2 25208.704} C_VEL
LIN {X 0,Y 680.458,Z 329.461,A -85,B 0,C 180,E1 25205.735,E2 25205.735} C_VEL
LIN {X 0,Y 680.46,Z 329.464,A -85,B 0,C 180,E1 25203.117,E2 25203.117} C_VEL
LIN {X 0,Y 680.502,Z 329.468,A -85,B 0,C 180,E1 25200.084,E2 25200.084} C_VEL
LIN {X 0,Y 680.443,Z 329.465,A -85,B 0,C 180,E1 25197.389,E2 25197.389} C_VEL
LIN {X 0,Y 680.463,Z 329.462,A -85,B 0,C 180,E1 25194.773,E2 25194.773} C_VEL
LIN {X 0,Y 680.457,Z 329.462,A -85,B 0,C 180,E1 25191.635,E2 25191.635} C_VEL
LIN {X 0,Y 680.432,Z 329.467,A -85,B 0,C 180,E1 25189.073,E2 25189.073} C_VEL
LIN {X 0,Y 680.486,Z 329.443,A -85,B 0,C 180,E1 25186.316,E2 25186.316} C_VEL
LIN {X 0,Y 680.437,Z 329.469,A -85,B 0,C 180,E1 25183.348,E2 25183.348} C_VEL
LIN {X 0,Y 680.42,Z 329.453,A -85,B 0,C 180,E1 25180.87,E2 25180.87} C_VEL
LIN {X 0,Y 680.472,Z 329.463,A -85,B 0,C 180,E1 25178.176,E2 25178.176} C_VEL
LIN {X 0,Y 680.425,Z 329.447,A -85,B 0,C 180,E1 25175.148,E2 25175.148} C_VEL
LIN {X 0,Y 680.422,Z 329.469,A -85,B 0,C 180,E1 25172.615,E2 25172.615} C_VEL
LIN {X 0,Y 680.524,Z 329.466,A -85,B 0,C 180,E1 25169.737,E2 25169.737} C_VEL
LIN {X 0,Y 680.435,Z 329.47,A -85,B 0,C 180,E1 25166.862,E2 25166.862} C_VEL
LIN {X 0,Y 680.439,Z 329.471,A -85,B 0,C 180,E1 25164.311,E2 25164.311} C_VEL
LIN {X 0,Y 680.499,Z 329.47,A -85,B 0,C 180,E1 25161.28,E2 25161.28} C_VEL
LIN {X 0,Y 680.465,Z 329.614,A -85,B 0,C 180,E1 25158.701,E2 25158.701} C_VEL
LIN {X 0,Y 681.565,Z 332.672,A -85,B 0,C 180,E1 25158.35,E2 25158.35} C_VEL
LIN {X 0,Y 682.707,Z 334.788,A -85,B 0,C 180,E1 25158.074,E2 25158.074} C_VEL
LIN {X 0,Y 688.542,Z 347.244,A -85,B 0,C 180,E1 25156.559,E2 25156.559} C_VEL
LIN {X 0,Y 690.589,Z 351.337,A -85,B 0,C 180,E1 25156.104,E2 25156.104} C_VEL
LIN {X 0,Y 698.327,Z 363.135,A -85,B 0,C 180,E1 25155.278,E2 25155.278} C_VEL
LIN {X 0,Y 700.808,Z 373.277,A -85,B 0,C 180,E1 25154.93,E2 25154.93} C_VEL
LIN {X 0,Y 698.428,Z 585.463,A -85,B 0,C 180,E1 25152.171,E2 25152.171} C_VEL
LIN {X 0,Y 696.118,Z 808.536,A -85,B 0,C 180,E1 25149.363,E2 25149.363} C_VEL
LIN {X 0,Y 695.54,Z 839.989,A -85,B 0,C 180,E1 25148.912,E2 25148.912} C_VEL
LIN {X 0,Y 694.786,Z 865.188,A -85,B 0,C 180,E1 25148.398,E2 25148.398} C_VEL
LIN {X 0,Y 693.901,Z 890.775,A -85,B 0,C 180,E1 25147.726,E2 25147.726} C_VEL
LIN {X 0,Y 692.785,Z 917.451,A -85,B 0,C 180,E1 25146.847,E2 25146.847} C_VEL
LIN {X 0,Y 691.791,Z 938.343,A -85,B 0,C 180,E1 25146.034,E2 25146.034} C_VEL
LIN {X 0,Y 690.754,Z 958.67,A -85,B 0,C 180,E1 25145.129,E2 25145.129} C_VEL
LIN {X 0,Y 689.673,Z 978.672,A -85,B 0,C 180,E1 25144.122,E2 25144.122} C_VEL
LIN {X 0,Y 688.522,Z 999.453,A -85,B 0,C 180,E1 25142.946,E2 25142.946} C_VEL
LIN {X 0,Y 687.068,Z 1024.24,A -85,B 0,C 180,E1 25141.35,E2 25141.35} C_VEL
LIN {X 0,Y 685.992,Z 1043.443,A -85,B 0,C 180,E1 25139.948,E2 25139.948} C_VEL
LIN {X 0,Y 684.975,Z 1061.817,A -85,B 0,C 180,E1 25138.464,E2 25138.464} C_VEL
LIN {X 0,Y 683.767,Z 1083.481,A -85,B 0,C 180,E1 25136.498,E2 25136.498} C_VEL
LIN {X 0,Y 682.982,Z 1099.688,A -85,B 0,C 180,E1 25134.845,E2 25134.845} C_VEL
